# B&R Automation Studio project EFI (part 9)

#### ArcLampGew.var - Local variables
```iecst
VAR CONSTANT
	MAXIMUM_QUANTITY_ALERTS : USINT := 6;
END_VAR
VAR
	data : REFERENCE TO ArcLampGew;
	Client : httpClient := (enable:=FALSE,send:=FALSE,abort:=FALSE,option:=0,pHost:=0,hostPort:=0,method:=httpMETHOD_GET,pUri:=0,pRequestHeader:=0,pRequestData:=0,requestDataLen:=0,pResponseHeader:=0,pResponseData:=0,responseDataSize:=0,pStatistics:=0,pStruct:=0,status:=0,tcpStatus:=0,httpStatus:=0,responseDataLen:=0,phase:=0,_i_state:=0,_i_result:=0,_ident:=0,_oldEnable:=0,_oldAbort:=0,_oldSend:=0,_state:=0,_internal:=0);
	ClientPost : httpClient := (enable:=FALSE,send:=FALSE,abort:=FALSE,option:=0,pHost:=0,hostPort:=0,method:=httpMETHOD_GET,pUri:=0,pRequestHeader:=0,pRequestData:=0,requestDataLen:=0,pResponseHeader:=0,pResponseData:=0,responseDataSize:=0,pStatistics:=0,pStruct:=0,status:=0,tcpStatus:=0,httpStatus:=0,responseDataLen:=0,phase:=0,_i_state:=0,_i_result:=0,_ident:=0,_oldEnable:=0,_oldAbort:=0,_oldSend:=0,_state:=0,_internal:=0);
	Doenable : BOOL := FALSE; (*Enables FUB Instance*)
	Dosend : BOOL := FALSE; (*Sends request on positive edge*)
	Host : STRING[100] := 'localhost';
	Responsedata : STRING[6000] := '';
	Ressource : STRING[80] := '';
	RequestHeader : httpResponseHeader_t;
	RequestHeaderPost : httpResponseHeader_t;
	credentialsFlat : STRING[80];
	CredentialsEncoder : httpEncodeBase64;
	credentialsBase64 : STRING[280];
	authenticationBase : STRING[180];
	strAux : STRING[80];
	JSON_Parse_0 : JSON_Parse;
	dataToParse : STRING[6000] := '';
	sysResp : SystemResp;
	LampsResp : AllLampsResp;
	UvLampsResp : UvStatusResp;
	alertsResp : AlertsLampResp;
	sysRespWrk : SystemResp;
	LampsRespWrk : AllLampsResp;
	UvLampsRespWrk : UvStatusResp;
	alertsRespWrk : AlertsLampResp;
	commsStatus : ArcLampGew_Comms := ARCLG_IDLE;
	commsStatus_copy : ArcLampGew_Comms := ARCLG_IDLE;
	xComsStatusChanged : BOOL;
	commsSubStatus : ArcLampGew_SubComms := ARCLGS_IDLE;
	dataDebug : STRING[1800];
	dataNotFound : STRING[180];
	CurrentState : ArcLampGew_State := ARCLGEW_NOT_INITIALIZED;
	CurrentState_copy : ArcLampGew_State := ARCLGEW_NOT_INITIALIZED;
	xCurrentStateChanged : BOOL;
END_VAR
VAR CONSTANT
	iHistoryLines : USINT := 25;
END_VAR
VAR
	StateHistory : ARRAY[0..iHistoryLines] OF ArcLampGew_State;
	iIndexHistory : USINT;
	iLamp : USINT;
	iAlert : USINT;
	CommsCmdReseted : CommsCommands;
	xAnyLampSelected : BOOL;
	xAnyLampInError : BOOL;
	tonErrorComms : TON;
	tonSendReadSystem : TON;
	tonDelaySendReadSystem : TON;
	resetedAlarms : ArcLampGew_Alarms;
	resetedAlarmsSummary : stEFI_AlarmSummary;
	resetedComsAlarms : ArcLampGew_CommsAlarms;
	xAuxVar : BOOL;
	iLampComs : USINT; (*Variable to define the lamp communicating with. NOT to use in loops*)
	iMaxLampSelected : USINT; (*The maximum selected lamp prepare to workwith*)
	paramURL : httpSetParamUrl;
	RequestDataPost : STRING[180];
	iStatusChanges : UINT;
	iReasonStop : UINT;
	iReasonCritical : UINT;
	iAnyAlarm : UINT;
	iAnyWarning : UINT;
	stEventLog : EventLog_typ;
	reasonSound : UINT;
	arCommsError : AutoResetSound;
	arLampInError1 : AutoResetSound;
	arLampInError2 : AutoResetSound;
	arJam : AutoResetSound;
	iTimesReadLamps : UINT;
	iTimesReadLampsUv : UINT;
	iTimesReadAlerts : UINT;
	iTimesResetAll : UINT;
	iTimesSelectLamp : UINT;
	iTimesDeselectLamp : UINT;
	iTimesStopSelected : UINT;
	iTimesStartSelected : UINT;
	iTimesDeselectAll : UINT;
	iTimesSetPower : UINT;
	iTimesReadSystem : UINT;
	iTimesCommsError : UINT;
	credentialsUser : STRING[80];
	credentialsUserInternal : STRING[80];
	strAuxCredentials : STRING[80];
	iSendClient : UINT;
	iSendPost : UINT;
	lastErrorReseted : ErrorWebServiceData;
	lastCommsError : ErrorWebServiceData;
END_VAR
VAR CONSTANT
	iHistoryCommsLines : USINT := 25;
END_VAR
VAR
	ErrorCommsHistory : ARRAY[0..iHistoryCommsLines] OF ErrorWebServiceData;
	iIndexCommsHistory : USINT;
	UvLampRespAssigWrk : REFERENCE TO UvLampResp;
	tonParsingError : TON;
	tonInputReady : TON;
	tonRetryCommand : TON;
	xResetNeeded : UINT;
	xReadSystemDelay : BOOL;
	iReasonToStop : USINT;
	resetedOuts : ArcLampGew_SignalsOut;
	resetedStatus : ArcLampGew_Status;
END_VAR
```

- Rhino API - Read-Write.postman_collection.json (not shown)

### ArcLampSim.typ
```iecst
TYPE
	ArcLampSimCommands_typ : 	STRUCT
		CreateError : BOOL;
	END_STRUCT;
	ArcLampSim_typ : 	STRUCT
		Commands : ArcLampSimCommands_typ;
	END_STRUCT;
END_TYPE
```

### Program Logical/ExtPack/_Cure/ArcLampGEW/ArcLampSim/ArcLampSim_v1/ArcLampSim (IEC)

#### ArcLampSim.var - Local variables
```iecst
VAR
	SimArcLamp : REFERENCE TO ArcLampSim_typ;
	dataArcLamp : REFERENCE TO ArcLampGew;
	tonTransport : TON;
	tonReady : TON;
	tonDry : TON;
	CommsCmdReseted : CommsCommands;
	tonCommand : TON;
	iIndexLamp : USINT;
	xSimulatingCommand : UINT;
	iSetLampTimes : UINT;
END_VAR
```

### CuringLed.typ
```iecst
TYPE
	CuringLedCheck_enum :
		(
		CHECK_INIT,
		CHECK_READ_CONFIG,
		CHECK_UPDATE_STATUS,
		CHECK_READY,
		CHECK_ERROR
		);
	CuringLedReadingLampUvTime_enum :
		(
		READINGUVTIME_NOT_INIT,
		READINGUVTIME_INIT,
		READINGUVTIME_READING,
		READINGUVTIME_READY,
		READINGUVTIME_ERROR
		);
	CuringLedReadingLampTemp_enum :
		(
		READINGTEMP_NOT_INIT,
		READINGTEMP_INIT,
		READINGTEMP_READING,
		READINGTEMP_READY,
		READINGTEMP_ERROR
		);
	CuringLedDetect_enum :
		(
		DETECTION_NOT_INIT,
		DETECTION_INIT,
		DETECTION_POLLING,
		DETECTION_SAVE_SERIAL_NUMBERS,
		DETECTION_FINISHING_POLLING,
		DETECTION_READ_INTENSITY,
		DETECTION_ASSIGN_POSITION,
		DETECTION_READY,
		DETECTION_ERROR
		);
	CuringLedConfig_enum :
		(
		CONFIGURATION_NOT_INIT,
		CONFIGURATION_INIT,
		CONFIGURATION_PREPARE_LAMP,
		CONFIGURATION_PREPARE_SLM,
		CONFIGURATION_SEND,
		CONFIGURATION_SENDING,
		CONFIGURATION_SENT,
		CONFIGURATION_READ,
		CONFIGURATION_READY
		);
	CuringLedStatus_enum :
		(
		CURINGLED_OFF,
		CURINGLED_INIT,
		CURINGLED_PREPARING,
		CURINGLED_READY,
		CURINGLED_EMITTING,
		CURINGLED_FAULTED
		);
	CuringLed_NitrogenStatus_enum :
		(
		CURINGNITRO_OFF,
		CURINGNITRO_INIT,
		CURINGNITRO_READY,
		CURINGNITRO_FAULT
		);
	CuringLed_ApplicationType_enum :
		( (*Defines application purpose of curing led. May be use to cure ink (white, color) or primer*)
		CURING_APP_UNDEFINED,
		CURING_APP_WHITE, (*White ink*)
		CURING_APP_COLOR, (*Any ink apart from white*)
		CURING_APP_PRIMER (*Varnish*)
		);
	CuringLed_Alarms_typ : 	STRUCT
		xChillerFaulted : BOOL;
		xN2HighFlow : BOOL;
		xN2LowFlow : BOOL;
		xCureSystemFaulted : BOOL; (*gui_q_xAlrOverallCureSystFaulted*)
		xLampsSlmNotConfigured : BOOL;
		xFrontDoorOpened : BOOL; (*Front door is opened. UV light is dangerous*)
		xPowerFailure : BOOL; (*Any power suppliy dc voltage has failed*)
		xSerialNumbersRepeated : BOOL; (*Some lamps has same serial number*)
		xSerialNumbersNotAssigned : BOOL; (*Any lamp has no serial number assigned*)
		xDetectionProcessFailed : BOOL; (*Serial number detection process has failed*)
		Lamps : ARRAY[0..MAX_LAST_CURING_LED_LAMP]OF CuringLed_Lamp_Alarms_typ;
	END_STRUCT;
	CuringLed_Lamp_Alarms_typ : 	STRUCT
		SLMFault : BOOL; (*SLM fault present on LED cure lamp*)
		ThermalFault : BOOL; (*Thermal fault present on LED cure lamp*)
		AnyWarning : BOOL; (*Warning if there is any not needed lamp in error.*)
		StatusFeedbackFault : BOOL; (*Slm status feedback from lamp missing in system status message*)
		xSlmWrongConfiguration : ARRAY[0..20]OF BOOL; (*SLM not configured properly*)
	END_STRUCT;
	CuringLed_Signals_In_typ : 	STRUCT
		xN2HighFlow : BOOL;
		xN2LowFlow : BOOL;
		xPsuDcOk : ARRAY[0..10]OF BOOL;
		xPsuAcOk : ARRAY[0..10]OF BOOL;
		xFrontDoorClosed : BOOL;
		xSafetyEnable : BOOL; (*The Enable signals are active. Do not show alarms related to this if not active*)
	END_STRUCT;
	CuringLed_Signals_Out_typ : 	STRUCT
		xPowerOnLamps : BOOL;
		xRunChiller : BOOL; (*Chiller has just one input named "Run"*)
		xPowerOnNitrogen : BOOL;
	END_STRUCT;
	CuringLed_Signals_typ : 	STRUCT
		Inputs : CuringLed_Signals_In_typ;
		Outputs : CuringLed_Signals_Out_typ;
	END_STRUCT;
	CuringLed_Comms_typ : 	STRUCT
		Ready : BOOL; (*To show the status of the startup process.*)
		ConfigOK : BOOL; (*Lamps SLMs configured*)
		Command : Comms_command_typ;
		Device : DeviceComms_typ;
	END_STRUCT;
	CuringLed_Status_typ : 	STRUCT
		xInstalled : BOOL;
		xEmitting : BOOL;
		DetectionState : CuringLedDetect_enum; (*State of the control*)
		Config : CuringLedConfig_enum; (*State of the control*)
		State : CuringLedStatus_enum; (*Status of the curing led: 0=off, 1=init, 2=ready, 3=emitting, 4=faulted*)
		NitroState : CuringLed_NitrogenStatus_enum;
		ChillerState : ChillerStatus_enum;
		iTotalNumSlms : UINT; (*Total number of slm of the curing bar*)
		xOptimizeCuring : BOOL; (*To cure just the document not the entire board*)
		xCureByStretch : BOOL; (*To configure lamps to cure by stretches*)
		xLampsDetected : BOOL; (*Active when all lamps installed have a serial number associated*)
		xLampsChecked : BOOL; (*Active when check of lamps current configuration match desired configuration*)
		xLampsConfigured : BOOL; (*Active when all lamps have been configured*)
		ManualCommands : CuringLed_ManualCommands_typ;
		iCuringAreaWidth : UINT;
		iCuringAreaOffsetL1 : INT;
		iCuringAreaOffsetL2 : INT;
	END_STRUCT;
	CuringLed_Parameters_typ : 	STRUCT
		xInstalled : BOOL;
		xEnabled : BOOL;
		iLampsQuantity : USINT; (*Total lamps in the CuringLed system. Max 16*)
		Mode : StGeneral_States_Mode;
		AutoMode : stEFI_MachineAutoModes;
		iChillerIndex : INT; (*Index of chiller used by the curing led lamp*)
		iCuringPosition : INT; (*Position of the led lamps bar in cm*)
		iCuringWindow : INT; (*Led lamps width in process direction (in mm). Depends on lamp's model. Alll lamps on same led bar have the same*)
		iDocumentWidth : UINT;
		iDocumentOffsetL1 : INT;
		iDocumentOffsetL2 : INT;
		iMaxCuringAreaWidth : UINT;
		iMaxCuringAreaOffsetL1 : INT;
		iMaxCuringAreaOffsetL2 : INT;
		iMediaWidth : UINT;
		iMediaOffsetL1 : INT;
		iMediaOffsetL2 : INT;
		xDoubleLine : BOOL;
		rBeltCurrentSpeed : REAL;
		rMinCureSpeed : REAL := 1;
		iPowerSuppliesQuantity : USINT; (*Total power supplies used to power all lamps in the curing led bar. Max 10*)
		xWhiteLedBar : BOOL; (*To set this variable to TRUE when curing led bar is used for white color*)
		xCureBySpeed : BOOL; (*Intensity of lamps set depending on machine speed*)
		xSimulationMode : BOOL;
		xOptimizeCuring : BOOL; (*Curing optimitzation required*)
		xCureByStretch : BOOL; (*Curing by stretch mode required*)
		xPhysicalTempFeedback : BOOL; (*When a plc card is installed to read temp from lamp using an AI*)
		iMappingBar : USINT;
		iSlmWidth : USINT := 25;
		CuringApplicationType : CuringLed_ApplicationType_enum;
	END_STRUCT;
	CuringLed_ManualCommands_typ : 	STRUCT
		xNitrogen : BOOL;
		DetectLamps : BOOL;
		ResetPSU : BOOL; (*Reset the PSU to power the Lamps*)
	END_STRUCT;
	CuringLed_Commands_typ : 	STRUCT
		PowerOn : BOOL;
		xDropPower : BOOL; (*Command to set lamps to a lower intensity than defined by curing mode or setpoint written by SW*)
		xRunNitrogenFlow : BOOL; (*Command to active nitrogen flow*)
		xUpdateTempValues : BOOL; (*Update temp values*)
		RunCuring : BOOL; (*When the media to cure is below the lamps*)
		Mute : BOOL; (*command xMute *)
		Reset : BOOL; (*command xReset*)
		Manual : CuringLed_ManualCommands_typ;
	END_STRUCT;
	CuringLed_typ : 	STRUCT
		Signals : CuringLed_Signals_typ;
		Commands : CuringLed_Commands_typ;
		Parameters : CuringLed_Parameters_typ;
		Status : CuringLed_Status_typ;
		Alarms : CuringLed_Alarms_typ;
		AlSummary : stEFI_AlarmSummary; (*Alarms Summary*)
		Comms : CuringLed_Comms_typ;
		Lamp : ARRAY[0..MAX_LAST_CURING_LED_LAMP]OF CuringLed_Lamp_typ;
		parSw : CuringLed_Sw_Parameters_typ;
	END_STRUCT;
	enComms_STEPS :
		(
		FRM_WAIT := 0, (*Defines the wait step*)
		FRM_OPEN := 10, (*Defines Step for FRM_xopen() *)
		FRM_CLEAR_BUFFER := 20, (*Defines Step for FRM_rbuf()*)
		FRM_PREPARE_SENDDATA := 21, (*Defines Step for preparing send data*)
		FRM_WRITE := 22, (*Defines Step for FRM_write()*)
		FRM_RELEASE_SEND_BUFFER := 23, (*Defines Step for FRM_robuf()*)
		FRM_READ := 30, (*Defines Step for FRM_read()*)
		FRM_COPY_RD_DATA := 31, (*Defines Step for storing read data*)
		FRM_RELEASE_READ_BUFFER := 32, (*Defines Step for FRM_rbuf()*)
		FRM_CLOSE := 40, (*Defines Step for FRM_close()*)
		FRM_ERROR := 255 (*Defines Step for Errorhandling*)
		);
	Comms_command_typ : 	STRUCT
		Open : BOOL; (*Open serial port and receive data*)
		Send : BOOL; (*Close serial port*)
		Receive : BOOL; (*Receive data from device*)
		Close : BOOL; (*Close serial port*)
	END_STRUCT;
	DeviceComms_typ : 	STRUCT
		step : enComms_STEPS := (0); (*Step of the Statemachine*)
		receive_data : STRING[800]; (*receive data*)
		send_data : STRING[80]; (*Send data*)
		FRM_xopen_0 : FRM_xopen; (*Functionblock FRM_xopen()*)
		xopenConfig : XOPENCONFIG; (*Configuration Type for FRM_xopen()*)
		FRM_gbuf_0 : FRM_gbuf; (*Functionblock FRM_gbuf()*)
		FRM_robuf_0 : FRM_robuf; (*Functionblock FRM_robuf()*)
		FRM_read_0 : FRM_read; (*Functionblock FRM_read()*)
		FRM_rbuf_0 : FRM_rbuf; (*Functionblock FRM_rbuf()*)
		FRM_write_0 : FRM_write; (*Functionblock FRM_write)*)
		FRM_close_0 : FRM_close; (*Functionblock FRM_close()*)
		DeviceName : STRING[22]; (*Devicename --> serial interface properties*)
	END_STRUCT;
	CuringLed_Lamp_typ : 	STRUCT
		Inputs : CuringLed_Lamp_Inputs_typ;
		Outputs : CuringLed_Lamp_Outputs_typ;
		Parameters : CuringLed_Lamp_Parameters_typ;
		Status : CuringLed_Lamp_Status_typ;
	END_STRUCT;
	CuringLed_Lamp_Status_typ : 	STRUCT
		stUvOnTimeRaw : STRING[10]; (*Total number of minutes that DC power has been applied*)
		rUvOnTime : REAL; (*Total number of minutes that DC power has been applied*)
		rTemp : REAL;
		stSerialNumber : STRING[6];
	END_STRUCT;
	CuringLed_Lamp_Parameters_typ : 	STRUCT
		xInstalled : BOOL := FALSE;
		EnabledByPosition : BOOL := TRUE; (*Enable lamp to be ready for curing depending on its position, board width and offsets*)
		iNumSLM : UINT; (*Number of stretches (slm) in this lamp*)
		iCuringLength : UINT; (*Length of lamp in mm. Per position in lamp's bar (length = cross direction)*)
		xSlmEnable : ARRAY[0..20]OF BOOL; (*SLM to be enabled for each lamp. 1:Must cure, 0: Must not cure*)
		xFullActive : BOOL;
		sSystemStatusFeedback : STRING[300];
		iFirstSlm : INT;
		iLastSlm : INT;
	END_STRUCT;
	CuringLed_Sw_Parameters_typ : 	STRUCT
		IntensitySetPoint : INT; (*Value of the Intensity in percentage. Minimum 10%. gui_i_iUvIntensitySetPointLed1*)
		xEnableDDC : BOOL; (*Enable the DDC functionality*)
		iPreCuringOffset : INT := 0; (*Pre curing offset set by SW in cm*)
		iPostCuringOffset : INT := 0; (*Post curing offset set by SW in cm*)
	END_STRUCT;
	CuringLed_Lamp_Inputs_typ : 	STRUCT
		TemperatureRaw : INT; (*Led temperature value in C.*)
		SLMFault : BOOL; (*SLM fault present on LED cure lamp 1*)
		ThermalFault : BOOL; (*Thermal fault present on LED cure lamp 1*)
	END_STRUCT;
	CuringLed_Lamp_Outputs_typ : 	STRUCT
		IntensityLampApplied : USINT; (*Value of the real intensity setpoint applied to lamp by the PLC*)
		IntensityLampRaw : INT; (*Value of the Intensity in Analog units*)
		EnableLamp : BOOL; (*Enable for each lamp of the curing LED*)
		rTemperature : REAL; (*Lamp  temperature value in C*)
		LampErrorCode : USINT;
		xSlmStatus : ARRAY[0..20]OF BOOL; (*SLM status. Shows SLM is active to cure: 1:On, 0:Off*)
	END_STRUCT;
END_TYPE
```

### CuringLed.var
```iecst
VAR
	iIndexCuringLed : USINT;
END_VAR
```

### Program Logical/ExtPack/_Cure/CuringLedCtrl/CuringLedCtrl_v1/CuringLedCtrl

#### CuringLedCtrlConstants.var
```iecst
VAR CONSTANT
	iSlmWidth : INT := 25;
	StCmdWrite : STRING[2] := 'w ';
	StOff : STRING[2] := 'Of';
	StValueDisableSlm : STRING[2] := ' 0';
	StValueEnableSlm : STRING[2] := ' 1';
	iMaxNumLamps : USINT := 16;
	StCmdEnableSlm : STRING[11] := ' slmenable ';
	StCheckIntensity : STRING[10] := ' intensity';
	StCmdRead : STRING[2] := 'r ';
	StDs : STRING[3] := ' ds';
	StCheckStatus : STRING[4] := ' son'; (*Check if UV is Enabled. [On = UV enabled, Off = UV disabled]*)
	StOn : STRING[2] := 'On';
	StMl : STRING[2] := 'm1';
	BUSY : UINT := 65535; (*Functionblock BUSY status*)
	StCmdDisableAll : STRING[9] := ' slmall 0';
	StCmdEnableAll : STRING[9] := ' slmall 1';
	rCureBySpeedWhiteIntercept : REAL := 14.84;
	rCureBySpeedDefaultIntercept : REAL := 0;
	rCureBySpeedWhiteSlope : REAL := 0.86;
	rCureBySpeedDefaultSlope : REAL := 1.67;
	rLampIntensitySlope : REAL := 327.67;
	StOk : STRING[2] := 'ok';
	StPoll : STRING[4] := 'poll';
	StIntensity : STRING[10] := ' intensity';
	StTemperature : STRING[4] := ' tmp';
	iMaxNumAttempts : INT := 2;
	MaxIntensityCuringBySpeed : USINT := 100;
	MinIntensityCuringBySpeed : USINT := 40;
END_VAR
VAR
	iIntensityAnswerLength : INT := 3;
	iStatusAnswerLength : INT := 2;
END_VAR
```

#### AlarmSound.st
```iecst
ACTION AlarmSound:

	// Alarms reseteable sound management.
	ars_AlrStop.xAlarm:= dataLed.AlSummary.xAlarmStop;
	ars_AlrStop.xSilence:= dataLed.Commands.Mute;
	ars_AlrStop();

	ars_AlrCritical.xAlarm:= dataLed.AlSummary.xAlarmCritical;
	ars_AlrCritical.xSilence:= dataLed.Commands.Mute;
	ars_AlrCritical();

	ars_AlrWarning.xAlarm:= dataLed.AlSummary.xAnyWarning;
	ars_AlrWarning.xSilence:= dataLed.Commands.Mute;
	ars_AlrWarning();

	dataLed.AlSummary.xAlarmSound:= //ars_AlrWarning.xAlarmSound OR
									ars_AlrStop.xAlarmSound OR
									ars_AlrCritical.xAlarmSound;

END_ACTION
```

#### CheckLampsConfig.st
```iecst
ACTION CheckLampsConfig:

	IF (xBoardPositionChanged OR dataLed.Alarms.xPowerFailure OR NOT dataLed.Commands.PowerOn OR EDGEPOS(xConfigurationFailed)) THEN
		CheckStep := CHECK_INIT;
	END_IF

	CASE CheckStep OF

		CHECK_INIT:
			IF dataLed.Status.xLampsConfigured THEN
				iIndexConfigLamps := 1;
				dataLed.Comms.Device.receive_data := '';
				FOR iIndexEraseReceivedData:=1 TO iLampsQuantity DO
					dataLed.Lamp[iIndexConfigLamps].Parameters.sSystemStatusFeedback := '';
				END_FOR
				CheckStep := CHECK_READ_CONFIG;
			END_IF

		CHECK_READ_CONFIG:
			//To set the message string
			ReadLampStatus;

			//To send command to lamp
			dataLed.Comms.Command.Send := TRUE;

			IF (dataLed.Comms.Device.receive_data <> '') THEN
				iSupplySide := 0;
				CheckStep := CHECK_UPDATE_STATUS;
			END_IF

		CHECK_UPDATE_STATUS:
			iNumLampSLM := dataLed.Lamp[iIndexConfigLamps].Parameters.iNumSLM; //Number of lamp's SLMs
			iMinBufferLength := 436 + iNumLampSLM*5; //DELOREAN-1923: Minimum buffer length when lamp gives all slm feedback is: 436+iNumLampSLM*5 (f.e: "1=On ")

			iSupplySide := FIND(dataLed.Comms.Device.receive_data, 'Supply Side');
			xValidStatusReading := iSupplySide>0;
			//IF dataLed.Comms.Device.FRM_read_0.buflng > 500(*iMinBufferLength*) THEN
			IF xValidStatusReading THEN
				iCheckStatusAttempts := 0;
				xSLMStatusRead := TRUE;

				//Saving slms status as lamp parameter
				FindInString := INT_TO_STRING(1);
				strcat(ADR(FindInString),ADR('='));
				iAnswerStringPosition := FIND(dataLed.Comms.Device.receive_data, FindInString);
				dataLed.Lamp[iIndexConfigLamps].Parameters.sSystemStatusFeedback := MID(dataLed.Comms.Device.receive_data, 280, iAnswerStringPosition);

				FOR iIndexConfigSlm:=1 TO iNumLampSLM DO
					CheckSlmStatus;
				END_FOR

				IF xSLMStatusRead THEN
					NextLamp;
				ELSE
					dataLed.Comms.Device.receive_data := '';
					CheckStep := CHECK_READ_CONFIG;
				END_IF

			ELSIF (iCheckStatusAttempts >= iMaxNumAttempts) THEN
				dataLed.Alarms.Lamps[iIndexConfigLamps].StatusFeedbackFault := TRUE;
				NextLamp;

			ELSIF dataLed.Comms.Device.step = FRM_WAIT THEN
				iCheckStatusAttempts := iCheckStatusAttempts + 1;
				dataLed.Comms.Device.receive_data := '';
				CheckStep := CHECK_READ_CONFIG;
			END_IF

		CHECK_READY:

	END_CASE

	dataLed.Comms.Device.send_data := StMessage; //To assign Message to dataled comms struct
	dataLed.Status.xLampsChecked := CheckStep = CHECK_READY;

END_ACTION

//Telegrams to be sent to curing led devices//
//To enable all slm in the lamp
ACTION ReadLampStatus:
	//To define the string to be sent to the lamp
	StMessage := StCmdRead;
	//strcat: Used to link (concat) several strings
	strcat(ADR(StMessage), ADR(dataLed.Lamp[iIndexConfigLamps].Status.stSerialNumber));
	strcat(ADR(StMessage), ADR(StMl));
	strcat(ADR(StMessage), ADR(StDs));
	//dataLed.Comms.Device.send_data := StMessage; //To assign Message to dataled comms struct

	iAnswerStringLength := 2;

	//This is the data received when reading status of a led. SLM status shown for a lamp with all SLM disabled:
	(*
	Product..........: Fire_Line_400_300, s/n 414086m1
	Firmware Ver.....: 01.02
	Log Entries......: 1020
	SLM Enables......:
	Supply Side 1=Off 2=Off 3=Off 4=Off 5=Off 6=Off 7=Off 8=Off 9=Off 10=Off 11=Off 12=Off Return Side
	SW-Disable Low.....: High
	SW-Enable High...: Low
	Global Control...: DB15
	Intensity........: 100
	Temperature......: 36.4
	Inputvolt........: 49.8
	Thermal Switch...: Enabled
	*)
END_ACTION

ACTION NextLamp:

	//Erasing buffer and going to next lamp
	iIndexConfigLamps := iIndexConfigLamps + 1;
	IF iIndexConfigLamps <= iLampsQuantity THEN
		dataLed.Comms.Device.receive_data := '';
		CheckStep := CHECK_READ_CONFIG;
	ELSE
		CheckStep := CHECK_READY;
	END_IF
END_ACTION

ACTION CheckSlmStatus:
	FindInString := INT_TO_STRING(iIndexConfigSlm);
	strcat(ADR(FindInString),ADR('='));
	iAnswerStringPosition := FIND(dataLed.Comms.Device.receive_data, FindInString);
	IF iIndexConfigSlm<10 THEN iAnswerStringPosition := iAnswerStringPosition+2; ELSE iAnswerStringPosition := iAnswerStringPosition+3; END_IF //X=On/Off
	StAnswer := MID(dataLed.Comms.Device.receive_data, iAnswerStringLength, iAnswerStringPosition);

	IF (StAnswer = StOn) THEN
		dataLed.Lamp[iIndexConfigLamps].Outputs.xSlmStatus[iIndexConfigSlm]:=TRUE;
	ELSIF (StAnswer = StOff) THEN
		dataLed.Lamp[iIndexConfigLamps].Outputs.xSlmStatus[iIndexConfigSlm]:=FALSE;
	ELSE
		xSLMStatusRead := FALSE;
	END_IF
END_ACTION
```

#### CheckParameters.st
```iecst
ACTION CheckParameters:

	iLampsQuantity := LIMIT(1,dataLed.Parameters.iLampsQuantity,iMaxNumLamps);
	iPowerSuppliesQuantity := LIMIT(1,dataLed.Parameters.iPowerSuppliesQuantity,6);

	FOR iIndexCuring:=1 TO iLampsQuantity DO
		dataLed.parSw.IntensitySetPoint:=LIMIT(10, dataLed.parSw.IntensitySetPoint, 100);
		dataLed.Lamp[iIndexCuring].Parameters.xInstalled := TRUE;
	END_FOR

	//Assigning parameters of curing area
	IF NOT dataLed.Status.xOptimizeCuring THEN
		dataLed.Status.iCuringAreaWidth := dataLed.Parameters.iMediaWidth;
		dataLed.Status.iCuringAreaOffsetL1 := dataLed.Parameters.iMediaOffsetL1;
		dataLed.Status.iCuringAreaOffsetL2 := dataLed.Parameters.iMediaOffsetL2;
	ELSE
		//Optimize curing will be active when EHD is enabled so plc does not have to consider metal bands overlap with to not burn it.
		//Document width has to be smaller than (MediaWidth- 2*Overlap). Document width is managed by SW
		dataLed.Status.iCuringAreaWidth := dataLed.Parameters.iDocumentWidth;
		dataLed.Status.iCuringAreaOffsetL1 := dataLed.Parameters.iDocumentOffsetL1;
		dataLed.Status.iCuringAreaOffsetL2 := dataLed.Parameters.iDocumentOffsetL2;
	END_IF

	dataLed.Status.iCuringAreaWidth := MIN(dataLed.Status.iCuringAreaWidth, dataLed.Parameters.iMaxCuringAreaWidth);
	dataLed.Status.iCuringAreaOffsetL1 := MAX(dataLed.Status.iCuringAreaOffsetL1, dataLed.Parameters.iMaxCuringAreaOffsetL1);
	dataLed.Status.iCuringAreaOffsetL2 := MIN(dataLed.Status.iCuringAreaOffsetL2, dataLed.Parameters.iMaxCuringAreaOffsetL2);

	//This action must be executed just once.
	IF iTotalNumSlms<=0 THEN
		//To sum all slm in the curing led bar. Depends on number of lamps and their width
		FOR iIndexEnableLamps:=1 TO iLampsQuantity DO
			dataLed.Lamp[iIndexEnableLamps].Parameters.iNumSLM := (dataLed.Lamp[iIndexEnableLamps].Parameters.iCuringLength/iSlmWidth);
			iTotalNumSlms :=  iTotalNumSlms + dataLed.Lamp[iIndexEnableLamps].Parameters.iNumSLM;
		END_FOR

		iTotalNumSlms :=  MIN(iTotalNumSlms, 100);
		dataLed.Status.iTotalNumSlms := iTotalNumSlms;
	END_IF

END_ACTION
```

#### CommsManager.st
```iecst
ACTION CommsManager:

	//To disable functions and open again when a READ command seems to be on hold to much time
	tonOpenPort.IN:= (dataLed.Comms.Device.step = FRM_READ);
	tonOpenPort.PT := T#10s;
	tonOpenPort();

	dataLed.Comms.Command.Open := tonOpenPort.Q;

	IF dataLed.Comms.Command.Open THEN																(*command for sender activation*)
		DisableFunctions;
		dataLed.Comms.Device.step := FRM_OPEN;

	ELSIF dataLed.Comms.Command.Close THEN															(*command for sender activation*)
		DisableFunctions;
		dataLed.Comms.Device.step := FRM_CLOSE;
	END_IF

	CASE dataLed.Comms.Device.step OF

		FRM_WAIT:
			IF dataLed.Comms.Command.Send THEN													(*command for sender activation*)
				dataLed.Comms.Device.step := FRM_OPEN;
			ELSIF dataLed.Comms.Command.Receive THEN											(*command for sender activation*)
				dataLed.Comms.Device.step := FRM_READ;
			END_IF

		FRM_OPEN:
			DisableFunctions;

			(*Parameters for FRM_xopen()*)
			dataLed.Comms.Device.FRM_xopen_0.enable := TRUE;

			dataLed.Comms.Device.FRM_xopen_0.device := ADR(dataLed.Comms.Device.DeviceName);
			dataLed.Comms.Device.FRM_xopen_0.mode := ADR('/PHY=RS485 /BD=57600 /DB=8 /PA=N /SB=1'); (*Modestring --> specifies the seria operation mode*)
			dataLed.Comms.Device.FRM_xopen_0.config := ADR(dataLed.Comms.Device.xopenConfig);		(*Additional Parameters, optional*)

			(*Additional Parameters for FRM_xopen()*)
			dataLed.Comms.Device.xopenConfig.idle := 10;											//Idle time between two characters
			dataLed.Comms.Device.xopenConfig.delimc := 0;											//activate two delimeters
			dataLed.Comms.Device.xopenConfig.delim[0] := 0; 										//CR - carridge return -> dec 13
			dataLed.Comms.Device.xopenConfig.delim[1] := 0; 										//LF - line feed -> dec 10
			dataLed.Comms.Device.xopenConfig.tx_cnt := 1;											//number of transmit buffers
			dataLed.Comms.Device.xopenConfig.rx_cnt := 1; 											//number of receive buffers
			dataLed.Comms.Device.xopenConfig.tx_len := 80; 											//length of transmit buffers
			dataLed.Comms.Device.xopenConfig.rx_len := 800; 										//lenght of receive buffers
			dataLed.Comms.Device.xopenConfig.argc := 0;												//activate additional options
			dataLed.Comms.Device.xopenConfig.argv := 0;												//parameters for additional options (check help)
			dataLed.Comms.Device.FRM_xopen_0();														//call the FRM_xopen() function

			xCommsOpened := dataLed.Comms.Device.FRM_xopen_0.status = 0;
			xOpeningComms := dataLed.Comms.Device.FRM_xopen_0.status = BUSY;

			IF dataLed.Comms.Device.FRM_xopen_0.status <> ERR_FUB_BUSY AND dataLed.Comms.Device.FRM_xopen_0.status <> ERR_FUB_ENABLE_FALSE THEN
				IF dataLed.Comms.Device.FRM_xopen_0.status = ERR_OK THEN
					dataLed.Comms.Device.step := FRM_CLEAR_BUFFER;
				ELSE
					dataLed.Comms.Device.step := FRM_ERROR;
				END_IF
			END_IF

		(*aquire sendbuffer for FRM_WRITE*)
		FRM_CLEAR_BUFFER:
			dataLed.Comms.Device.FRM_gbuf_0.enable := TRUE;
			dataLed.Comms.Device.FRM_gbuf_0.ident := dataLed.Comms.Device.FRM_xopen_0.ident;
			dataLed.Comms.Device.FRM_gbuf_0();																	(*call the FRM_gbuf() function*)

			xBufferCleared := dataLed.Comms.Device.FRM_gbuf_0.status = 0;
			xClearingBuffer := dataLed.Comms.Device.FRM_gbuf_0.status = BUSY;

			IF dataLed.Comms.Device.FRM_gbuf_0.status <> ERR_FUB_BUSY AND dataLed.Comms.Device.FRM_gbuf_0.status <> ERR_FUB_ENABLE_FALSE THEN
				IF dataLed.Comms.Device.FRM_gbuf_0.status = ERR_OK THEN
					memset(dataLed.Comms.Device.FRM_gbuf_0.buffer,0,dataLed.Comms.Device.FRM_gbuf_0.buflng);		//clear sendbuffer
					dataLed.Comms.Device.step := FRM_PREPARE_SENDDATA;
				ELSE
					dataLed.Comms.Device.step := FRM_ERROR;
				END_IF
			END_IF

		(*prepare senddata, copy data to sendbuffer*)
		FRM_PREPARE_SENDDATA:
			send_data := dataLed.Comms.Device.send_data;
			strcat(ADR(send_data),ADR('$R$L'));
			strcpy(dataLed.Comms.Device.FRM_gbuf_0.buffer,ADR(send_data));					(*copy senddata to sendbuffer*)

			dataLed.Comms.Device.step := FRM_WRITE;																(*--> next step*)

		(*write data to interface*)
		FRM_WRITE:
			(*Parameters for FRM_write()*)
			dataLed.Comms.Device.FRM_write_0.enable := TRUE;
			dataLed.Comms.Device.FRM_write_0.ident := dataLed.Comms.Device.FRM_xopen_0.ident;					(*ident from FRM_xopen()*)
			dataLed.Comms.Device.FRM_write_0.buffer := dataLed.Comms.Device.FRM_gbuf_0.buffer;					(*sendbuffer*)
			dataLed.Comms.Device.FRM_write_0.buflng := strlen(ADR(send_data));								(*net length of senddata*)

			dataLed.Comms.Device.FRM_write_0();																	(*call the FRM_write() function*)

			xBufferSent := dataLed.Comms.Device.FRM_write_0.status = 0;
			xSendingBuffer := dataLed.Comms.Device.FRM_write_0.status = BUSY;

			IF dataLed.Comms.Device.FRM_write_0.status <> ERR_FUB_BUSY AND dataLed.Comms.Device.FRM_write_0.status <> ERR_FUB_ENABLE_FALSE THEN
				IF dataLed.Comms.Device.FRM_write_0.status = ERR_OK THEN
					dataLed.Comms.Device.step := FRM_RELEASE_SEND_BUFFER;
				ELSE
					dataLed.Comms.Device.step := FRM_ERROR;
				END_IF
			END_IF

		(*release sendbuffer in case of no successful write operation*)
		FRM_RELEASE_SEND_BUFFER:
			dataLed.Comms.Device.FRM_robuf_0.enable := TRUE;
			dataLed.Comms.Device.FRM_robuf_0.buffer := dataLed.Comms.Device.FRM_gbuf_0.buffer;					(*sendbuffer*)
			dataLed.Comms.Device.FRM_robuf_0.buflng := dataLed.Comms.Device.FRM_gbuf_0.buflng;					(*buffer length*)
			dataLed.Comms.Device.FRM_robuf_0.ident := dataLed.Comms.Device.FRM_xopen_0.ident;					(*ident open*)
			dataLed.Comms.Device.FRM_robuf_0();																	(*call the FRM_robuf() function*)

			xBufferSendReleased := dataLed.Comms.Device.FRM_robuf_0.status = 0;
			xReleasingSendBuffer := dataLed.Comms.Device.FRM_robuf_0.status = BUSY;

			IF dataLed.Comms.Device.FRM_robuf_0.status <> ERR_FUB_BUSY AND dataLed.Comms.Device.FRM_robuf_0.status <> ERR_FUB_ENABLE_FALSE THEN
				IF dataLed.Comms.Device.FRM_robuf_0.status = ERR_OK THEN
					dataLed.Comms.Device.step := FRM_READ;
				ELSE
					dataLed.Comms.Device.step := FRM_ERROR;
				END_IF
			END_IF

		(*read data from serial interface*)
		FRM_READ:
			dataLed.Comms.Device.FRM_read_0.enable := TRUE;
			dataLed.Comms.Device.FRM_read_0.ident := dataLed.Comms.Device.FRM_xopen_0.ident;
			dataLed.Comms.Device.FRM_read_0();																	(*call the FRM_read() function*)

			xBufferRead := dataLed.Comms.Device.FRM_read_0.status = 0;
			xReadBufferNoInput := dataLed.Comms.Device.FRM_read_0.status = frmERR_NOINPUT;
			xReadBufferInputError := dataLed.Comms.Device.FRM_read_0.status = frmERR_INPUTERROR;

			IF dataLed.Comms.Device.FRM_read_0.status <> ERR_FUB_BUSY AND dataLed.Comms.Device.FRM_read_0.status <> ERR_FUB_ENABLE_FALSE THEN
				IF dataLed.Comms.Device.FRM_read_0.status = ERR_OK THEN
					dataLed.Comms.Device.step := FRM_COPY_RD_DATA;
				ELSIF  dataLed.Comms.Device.FRM_read_0.status = frmERR_NOINPUT THEN
					dataLed.Comms.Device.step := FRM_READ;
				ELSIF dataLed.Comms.Device.FRM_read_0.status = frmERR_INPUTERROR THEN
					dataLed.Comms.Device.step := FRM_RELEASE_READ_BUFFER;
				ELSE
					dataLed.Comms.Device.step := FRM_ERROR;
				END_IF
			END_IF

		(*copy data out of the receive buffer*)
		FRM_COPY_RD_DATA:
			memset(ADR(dataLed.Comms.Device.receive_data),0,SIZEOF(dataLed.Comms.Device.receive_data));										(*clear read_data buffer*)
			memcpy(ADR(dataLed.Comms.Device.receive_data),dataLed.Comms.Device.FRM_read_0.buffer,dataLed.Comms.Device.FRM_read_0.buflng);   (*copy and evaluate read data*)
			dataLed.Comms.Device.step := FRM_RELEASE_READ_BUFFER;																			(*release read buffer*)

		(*release readbuffer*)
		FRM_RELEASE_READ_BUFFER:
			(*Parameters for FRM_rbuf()*)
			dataLed.Comms.Device.FRM_rbuf_0.enable := TRUE;
			dataLed.Comms.Device.FRM_rbuf_0.ident := dataLed.Comms.Device.FRM_xopen_0.ident;					(*ident from FRM_xopen()*)
			dataLed.Comms.Device.FRM_rbuf_0.buffer := dataLed.Comms.Device.FRM_read_0.buffer;					(*read buffer*)
			dataLed.Comms.Device.FRM_rbuf_0.buflng := dataLed.Comms.Device.FRM_read_0.buflng;					(*length of sendbuffer*)
			dataLed.Comms.Device.FRM_rbuf_0();																	(*call the FRM_rbuf() function*)

			xBufferReadReleased := dataLed.Comms.Device.FRM_rbuf_0.status = 0;
			xReleasingReadBuffer := dataLed.Comms.Device.FRM_rbuf_0.status = BUSY;
			xBufferReadInvalid := dataLed.Comms.Device.FRM_rbuf_0.status = frmERR_INVALIDBUFFER;

			IF dataLed.Comms.Device.FRM_rbuf_0.status <> ERR_FUB_BUSY AND dataLed.Comms.Device.FRM_rbuf_0.status <> ERR_FUB_ENABLE_FALSE THEN
				IF dataLed.Comms.Device.FRM_rbuf_0.status = ERR_OK THEN
					dataLed.Comms.Device.step := FRM_CLOSE;
				ELSIF dataLed.Comms.Device.FRM_rbuf_0.status = frmERR_INVALIDBUFFER THEN
					dataLed.Comms.Device.step := FRM_READ;
				ELSE
					dataLed.Comms.Device.step := FRM_ERROR;
				END_IF
			END_IF

		(*close the interface*)
		FRM_CLOSE:
			DisableFunctions;

			dataLed.Comms.Device.FRM_close_0.enable := TRUE;
			dataLed.Comms.Device.FRM_close_0.ident := dataLed.Comms.Device.FRM_xopen_0.ident;	(*ident from FRM_xopen()*)
			dataLed.Comms.Device.FRM_close_0();													(*call the FRM_close() function*)

			xCommsClosed := dataLed.Comms.Device.FRM_close_0.status = 0;
			xClosingComms := dataLed.Comms.Device.FRM_close_0.status = BUSY;

			IF dataLed.Comms.Device.FRM_close_0.status <> ERR_FUB_BUSY AND dataLed.Comms.Device.FRM_close_0.status <> ERR_FUB_ENABLE_FALSE THEN
				IF dataLed.Comms.Device.FRM_close_0.status = ERR_OK THEN
					dataLed.Comms.Device.step := FRM_WAIT;
				ELSE
					dataLed.Comms.Device.step := FRM_ERROR;
				END_IF
			END_IF

		(*error handling*)
		FRM_ERROR:
			DisableFunctions;
			dataLed.Comms.Device.step := FRM_WAIT;  (*not implementet yet, check help for error codes*)

	END_CASE

	//Store the history OF the error code TO easy the debug
	IF dataLed.Comms.Device.step<>StateHistory[0] THEN
		FOR iIndexHistory:=iHistoryLines TO 1 BY -1 DO
			StateHistory[iIndexHistory]:=StateHistory[iIndexHistory-1];
		END_FOR
		StateHistory[0]:=dataLed.Comms.Device.step;
	END_IF

	//Comms commands
	dataLed.Comms.Command := CommsCommandsReset;

END_ACTION

ACTION DisableFunctions:
	dataLed.Comms.Device.FRM_close_0.enable := FALSE;
	dataLed.Comms.Device.FRM_gbuf_0.enable := FALSE;
	dataLed.Comms.Device.FRM_rbuf_0.enable := FALSE;
	dataLed.Comms.Device.FRM_read_0.enable := FALSE;
	dataLed.Comms.Device.FRM_robuf_0.enable := FALSE;
	dataLed.Comms.Device.FRM_write_0.enable := FALSE;
	dataLed.Comms.Device.FRM_xopen_0.enable := FALSE;
END_ACTION
```

#### ConfigureLamps.st
```iecst
ACTION ConfigureLamps:

	IF dataLed.Alarms.xPowerFailure OR NOT dataLed.Commands.PowerOn THEN ConfigCtrl := CONFIGURATION_NOT_INIT; END_IF
	IF xBoardPositionChanged OR EDGEPOS(xConfigurationFailed) THEN ConfigCtrl := CONFIGURATION_INIT; END_IF

	CASE ConfigCtrl OF

		CONFIGURATION_NOT_INIT:

		CONFIGURATION_INIT:
			iIndexConfigLamps := 1;
			iIndexConfigSlm := 0;
			ConfigCtrl := CONFIGURATION_PREPARE_LAMP;

		CONFIGURATION_PREPARE_LAMP:
			//To evaluate only lamps that are going to be active (EnabledByPosition)
			IF NOT dataLed.Lamp[iIndexConfigLamps].Parameters.EnabledByPosition THEN
				DisableAllSlm;
			ELSE
				//To enable all SLM by default
				EnableAllSlm;
			END_IF
			ConfigCtrl := CONFIGURATION_SEND;

		CONFIGURATION_PREPARE_SLM:
			iNumLampSLM := dataLed.Lamp[iIndexConfigLamps].Parameters.iNumSLM; //Number of lamp's SLMs
			IF iIndexConfigSlm<=iNumLampSLM THEN
				//An active lamp might be full used or just use some SLMs
				IF (NOT dataLed.Lamp[iIndexConfigLamps].Parameters.xSlmEnable[iIndexConfigSlm]) THEN
					StIndex := INT_TO_STRING(iIndexConfigSlm);
					DisableSlm;
				END_IF
				ConfigCtrl := CONFIGURATION_SEND;
			ELSE
				iIndexConfigSlm := 0; //1;
				ConfigCtrl := CONFIGURATION_SENT;
			END_IF

		CONFIGURATION_SEND:
			dataLed.Comms.Command.Send := TRUE;
			ConfigCtrl := CONFIGURATION_SENDING;

		CONFIGURATION_SENDING:
			IF (StAnswer = StGoodAnswer) THEN
				IF (dataLed.Lamp[iIndexConfigLamps].Parameters.xFullActive OR NOT dataLed.Lamp[iIndexConfigLamps].Parameters.EnabledByPosition) THEN
					ConfigCtrl := CONFIGURATION_SENT;
				ELSE
					ConfigCtrl := CONFIGURATION_PREPARE_SLM;
					iIndexConfigSlm := iIndexConfigSlm + 1;
				END_IF
				dataLed.Comms.Device.receive_data := '';
			ELSIF dataLed.Comms.Device.step = FRM_WAIT THEN
				ConfigCtrl := CONFIGURATION_SEND;
			END_IF

		CONFIGURATION_SENT:
			iIndexConfigLamps := iIndexConfigLamps + 1;
			IF iIndexConfigLamps > iLampsQuantity THEN
				ConfigCtrl := CONFIGURATION_READY;
			ELSE
				ConfigCtrl := CONFIGURATION_PREPARE_LAMP;
			END_IF

		CONFIGURATION_READY:

	END_CASE

	dataLed.Comms.Device.send_data := StMessage; //To assign Message to dataled comms struct
	StAnswer := MID(dataLed.Comms.Device.receive_data, iAnswerStringLength, iAnswerStringPosition);
	dataLed.Status.xLampsConfigured := ConfigCtrl = CONFIGURATION_READY;
	dataLed.Status.Config := ConfigCtrl;

END_ACTION

//Telegrams to be sent to curing led devices//
//To enable all slm in the lamp
ACTION EnableAllSlm:
	//To define the string to be sent to the lamp
	StMessage := StCmdWrite;
	//strcat: Used to link (concat) several strings
	strcat(ADR(StMessage), ADR(dataLed.Lamp[iIndexConfigLamps].Status.stSerialNumber));
	strcat(ADR(StMessage), ADR(StMl));
	strcat(ADR(StMessage), ADR(StCmdEnableAll));

	//Devices answers "ok"
	StGoodAnswer := StOk;
	iAnswerStringPosition := 1;
	iAnswerStringLength := 2;
END_ACTION

//To disable all slm in the lamp
ACTION DisableAllSlm:
	//To define the string to be sent to the lamp
	StMessage := StCmdWrite;
	//strcat: Used to link (concat) several strings
	strcat(ADR(StMessage), ADR(dataLed.Lamp[iIndexConfigLamps].Status.stSerialNumber));
	strcat(ADR(StMessage), ADR(StMl));
	strcat(ADR(StMessage), ADR(StCmdDisableAll));

	//Devices answers "ok"
	StGoodAnswer := StOk;
	iAnswerStringPosition := 1;
	iAnswerStringLength := 2;
END_ACTION

//To enable an specific slm in the lamp
ACTION EnableSlm:
	//To define the string to be sent to the lamp
	StMessage := StCmdWrite;
	//strcat: Used to link (concat) several strings
	strcat(ADR(StMessage), ADR(dataLed.Lamp[iIndexConfigLamps].Status.stSerialNumber));
	strcat(ADR(StMessage), ADR(StMl));
	strcat(ADR(StMessage), ADR(StCmdEnableSlm));
	strcat(ADR(StMessage), ADR(StIndex));
	strcat(ADR(StMessage), ADR(StValueEnableSlm));

	//Device answers "SLMxx=On" when DisableSlm command is sent, where xx is SLM Index, so:
	StGoodAnswer := StOn;
	IF iIndexConfigSlm<10 THEN iAnswerStringPosition := 6; ELSE iAnswerStringPosition := 7; END_IF
	iAnswerStringLength := 2;
END_ACTION

//To disable an specific slm in the lamp
ACTION DisableSlm:
	//To define the string to be sent to the lamp
	StMessage := StCmdWrite;
	//strcat: Used to link (concat) several strings
	strcat(ADR(StMessage), ADR(dataLed.Lamp[iIndexConfigLamps].Status.stSerialNumber));
	strcat(ADR(StMessage), ADR(StMl));
	strcat(ADR(StMessage), ADR(StCmdEnableSlm));
	strcat(ADR(StMessage), ADR(StIndex));
	strcat(ADR(StMessage), ADR(StValueDisableSlm));

	//Device answers "SLMxx=Off" when DisableSlm command is sent, where xx is SLM Index, so:
	StGoodAnswer := StOff;
	IF iIndexConfigSlm<10 THEN iAnswerStringPosition := 6; ELSE iAnswerStringPosition := 7; END_IF
	iAnswerStringLength := 2;
END_ACTION
```

#### EnableLamps.st
```iecst
ACTION EnableLamps:
	//Enabling lamps to be activated depending on media width, offset register and line mode (single or 2up)
	iLampPosition := 0;

		IF NOT dataLed.Parameters.xDoubleLine THEN

			//							FEEDER/PRIMER						//
			//																//
			//////////////////////////////////////////////////////////////////
			//User side											//Back side //
			//					  											//
			//								"N" iLampPosition				//
			//----------------------------------------------->|				//
			//[[	1 	  ]][[	...	 ]][[	...	 ]][[	...	 ]][[	 N 	 ]]	//
			//			   ||		  ||	 0	  ||		  ||			//
			//					  			 |								//
			//					  			 |								//
			//			OffsetL1(-)<---------|--------->(+)					//
			//			////////////////////////////////////////////		//
			//			////////////////////////////////////////////		//
			//			////////////////////////////////////////////		//
			//			////////////////////////////////////////////		//
			//			////////////////////////////////////////////		//
			//			////////////////////////////////////////////		//
			//			////////////////////////////////////////////		//
			//			////////////////////////////////////////////		//
			//			|<-------		MediaWidth			------>|		//
			//								 								//
			//iBoardInitPos													//
			//--------->|													//
			//									iBoardFinalPosition			//
			//---------------------------------------------------->|		//
			//////////////////////////////////////////////////////////////////
			//																//
			//							DRYER/STACKER						//

			iBoardInitPosition := MAX(0, iCenterPosition + dataLed.Status.iCuringAreaOffsetL1);
			iBoardFinalPosition := MIN(iTotalWidth, iBoardInitPosition + dataLed.Status.iCuringAreaWidth);
			FOR iIndexEnableLamps:=1 TO iLampsQuantity DO
				iLampPosition := iLampPosition + dataLed.Lamp[iIndexEnableLamps-1].Parameters.iCuringLength;
				dataLed.Lamp[iIndexEnableLamps].Parameters.EnabledByPosition := (iBoardInitPosition < (iLampPosition + dataLed.Lamp[iIndexEnableLamps].Parameters.iCuringLength)) AND
																				(iLampPosition < iBoardFinalPosition);
			END_FOR

		ELSE
			//							FEEDER/PRIMER						//
			//																//
			//////////////////////////////////////////////////////////////////
			//User side											//Back side //
			//					  											//
			//								"N" iLampPosition				//
			//----------------------------------------------->|				//
			//[[	1 	  ]][[	...	 ]][[	...	 ]][[	...	 ]][[	 N 	 ]]	//
			//			   ||		  ||	0	  ||		  ||			//
			//		/////////////////		|	/////////////////			//
			//		/////////////////		|	/////////////////			//
			//		/////////////////		|	/////////////////			//
			//		/////////////////		|	/////////////////			//
			//		/////////////////		|	/////////////////			//
			//		/////////////////		|	/////////////////			//
			//		/////////////////		|	/////////////////			//
			//		/////////////////		|	/////////////////			//
			//		|<- MediaWidth->|		|	|<- MediaWidth->|			//
			//								|								//
			//	iRegisterOffsetL1(-)|<------|-->|iRegisterOffsetL2(+)		//
			//								|								//
			//																//
			//iBoardInitPos													//
			//----->|														//
			//								iBoardFinalPosition				//
			//-------------------------------------------------->|			//
			//								 								//
			//////////////////////////////////////////////////////////////////
			//																//
			//							DRYER/STACKER						//

			iBoardInitPosition := MAX(0,iCenterPosition + dataLed.Status.iCuringAreaOffsetL1);
			iBoardFinalPosition := MIN(iTotalWidth, iCenterPosition + dataLed.Status.iCuringAreaOffsetL2 + dataLed.Status.iCuringAreaWidth);
			FOR iIndexEnableLamps:=1 TO iLampsQuantity DO
				iLampPosition := iLampPosition + dataLed.Lamp[iIndexEnableLamps-1].Parameters.iCuringLength;
				dataLed.Lamp[iIndexEnableLamps].Parameters.EnabledByPosition := (iBoardInitPosition < (iLampPosition + dataLed.Lamp[iIndexEnableLamps].Parameters.iCuringLength)) AND
																				(iLampPosition<iBoardFinalPosition);
			END_FOR

		END_IF

END_ACTION

ACTION MemoBoardParameters:
	iPreviousWidth := dataLed.Status.iCuringAreaWidth;
	iPreviousOffsetRegisterL1 := dataLed.Status.iCuringAreaOffsetL1;
	iPreviousOffsetRegisterL2 := dataLed.Status.iCuringAreaOffsetL2;
END_ACTION
```

#### LedsCuringWidthCalculation.st
```iecst
ACTION StretchesCalculation:

	//Disabling all curing led bar's SLMs
	FOR iIndexEnableSlm:=0 TO iTotalNumSlms DO
		xCuringLedSlms[iIndexEnableSlm] := FALSE;
	END_FOR

	//DELOREAN-1778: To set printer's center
	iTotalWidth := iTotalNumSlms*iSlmWidth;
	iCenterPosition := REAL_TO_INT(iTotalWidth/2);

END_ACTION

ACTION SingleLineCalculation:
	//To caculate first SLM of the total curing led bar SLMs
	rFirstCuringBarSlmL1 := INT_TO_REAL(iCenterPosition + dataLed.Status.iCuringAreaOffsetL1)/iSlmWidth;
	pInteger := ADR(rInteger);
	rMantissa := modf(rFirstCuringBarSlmL1, pInteger);

	iFirstCuringBarSlmL1 := REAL_TO_UINT(rFirstCuringBarSlmL1);
	IF rMantissa = 0.0 THEN iFirstCuringBarSlmL1 := iFirstCuringBarSlmL1 + 1; END_IF

	//To caculate last SLM of the total curing led bar SLMs
	rLastCuringBarSlmL1 := (UINT_TO_REAL(iCenterPosition + dataLed.Status.iCuringAreaOffsetL1 + dataLed.Status.iCuringAreaWidth)/INT_TO_REAL(iSlmWidth));
	pInteger := ADR(rInteger);
	rMantissa := modf(rLastCuringBarSlmL1, pInteger);

	iLastCuringBarSlmL1 := REAL_TO_UINT(rInteger);
	IF rMantissa > 0.0 THEN iLastCuringBarSlmL1 := iLastCuringBarSlmL1 + 1; END_IF
	iLastCuringBarSlmL1 := LIMIT(iFirstCuringBarSlmL1, iLastCuringBarSlmL1, iTotalNumSlms);

	//Activating curing led bar's SLMs
	FOR iIndexEnableSlm:=iFirstCuringBarSlmL1 TO iLastCuringBarSlmL1 DO
		xCuringLedSlms[iIndexEnableSlm] := TRUE;
	END_FOR

	//To enable lamps stretches
	iLastLampSLM := 0;
	FOR iIndexEnableLamps:=1 TO iLampsQuantity DO
		iNumLampSLM := dataLed.Lamp[iIndexEnableLamps].Parameters.iNumSLM; //Number of lamp's SLMs

		//Lamp's first SLM of array "xCuringLedSlms" which considers all SLM in the curing led bar
		iFirstLampSLM := iLastLampSLM + 1;
		iLastLampSLM := iLastLampSLM + dataLed.Lamp[iIndexEnableLamps].Parameters.iNumSLM;

		dataLed.Lamp[iIndexEnableLamps].Parameters.iFirstSlm := iFirstLampSLM;
		dataLed.Lamp[iIndexEnableLamps].Parameters.iLastSlm := iLastLampSLM;

		dataLed.Lamp[iIndexEnableLamps].Parameters.xFullActive := TRUE;

		//Calculating slm mirrored to indexSlm. So xCuringLedSlms starts counting from user side to drive side. But lamps are mechanically assemblied in a reverse way, here an image to understand:

		//xCuringLedSlms[x]	  1						  14  15					  28  29					  42  43					  56
		//Lamp's slm index	  14					   1  14					   1  14					   1  14					   1
							//							//							//							//							//
		//FRONT/USER SIDE//	//			1				//			2				//			3				//			4				//		//REAR/WALKWAY SIDE//
							//							//							//							//							//
							//////////////////////////////////////////////////////////////////////////////////////////////////////////////////

		FOR iIndexEnableSlm:=1 TO iNumLampSLM DO
			iMirrorSlm := iLastLampSLM - iIndexEnableSlm + 1;
			dataLed.Lamp[iIndexEnableLamps].Parameters.xSlmEnable[iIndexEnableSlm] := xCuringLedSlms[iMirrorSlm];

			IF (NOT dataLed.Lamp[iIndexEnableLamps].Parameters.xSlmEnable[iIndexEnableSlm]) THEN
				dataLed.Lamp[iIndexEnableLamps].Parameters.xFullActive := FALSE;
			END_IF
		END_FOR
	END_FOR

END_ACTION

ACTION DoubleLineCalculation:

	///////////		L1		///////////
	rFirstCuringBarSlmL1 := INT_TO_REAL(iCenterPosition + dataLed.Status.iCuringAreaOffsetL1)/iSlmWidth;
	iFirstCuringBarSlmL1 := REAL_TO_UINT(rFirstCuringBarSlmL1) + 1;

	//To caculate last SLM of the total curing led bar SLMs
	rLastCuringBarSlmL1 := (UINT_TO_REAL(iCenterPosition + dataLed.Status.iCuringAreaOffsetL1 + dataLed.Status.iCuringAreaWidth)/INT_TO_REAL(iSlmWidth));
	pInteger := ADR(rInteger);
	rMantissa := modf(rLastCuringBarSlmL1, pInteger);

	iLastCuringBarSlmL1 := REAL_TO_UINT(rInteger);
	IF rMantissa > 0.0 THEN iLastCuringBarSlmL1 := iLastCuringBarSlmL1 + 1; END_IF
	iLastCuringBarSlmL1 := LIMIT(iFirstCuringBarSlmL1, iLastCuringBarSlmL1, REAL_TO_UINT(iTotalNumSlms/2));

	//Activating curing led bar's SLMs
	FOR iIndexEnableSlm:=iFirstCuringBarSlmL1 TO iLastCuringBarSlmL1 DO
		xCuringLedSlms[iIndexEnableSlm] := TRUE;
	END_FOR

	///////////		L2		///////////
	//To caculate first SLM of the total curing led bar SLMs
	rFirstCuringBarSlmL2 := (UINT_TO_REAL(iCenterPosition + dataLed.Status.iCuringAreaOffsetL2)/INT_TO_REAL(iSlmWidth));
	pInteger := ADR(rInteger);
	rMantissa := modf(rFirstCuringBarSlmL2, pInteger);

	iFirstCuringBarSlmL2 := REAL_TO_UINT(rInteger);
	IF rMantissa > 0.0 THEN iFirstCuringBarSlmL2 := iFirstCuringBarSlmL2 + 1; END_IF
	iFirstCuringBarSlmL2 := LIMIT(iLastCuringBarSlmL1, iFirstCuringBarSlmL2, iTotalNumSlms);

	//To caculate last SLM of the total curing led bar SLMs
	rLastCuringBarSlmL2 := (INT_TO_REAL(iCenterPosition + dataLed.Status.iCuringAreaOffsetL2 + dataLed.Status.iCuringAreaWidth)/INT_TO_REAL(iSlmWidth));
	pInteger := ADR(rInteger);
	rMantissa := modf(rLastCuringBarSlmL2, pInteger);

	iLastCuringBarSlmL2 := REAL_TO_UINT(rInteger);
	IF rMantissa > 0.0 THEN iLastCuringBarSlmL2 := iLastCuringBarSlmL2 + 1; END_IF
	iLastCuringBarSlmL2 := LIMIT(iFirstCuringBarSlmL2, iLastCuringBarSlmL2, iTotalNumSlms);

	FOR iIndexEnableSlm:=iFirstCuringBarSlmL2 TO iLastCuringBarSlmL2 DO
		xCuringLedSlms[iIndexEnableSlm] := TRUE;
	END_FOR

	///////////		To enable lamps stretches		///////////
	iLastLampSLM := 0;
	FOR iIndexEnableLamps:=1 TO iLampsQuantity DO
		iNumLampSLM := dataLed.Lamp[iIndexEnableLamps].Parameters.iNumSLM; //Number of lamp's SLMs

		//Lamp's first SLM of array "xCuringLedSlms" which considers all SLM in the curing led bar
		iFirstLampSLM := iLastLampSLM + 1;
		iLastLampSLM := iLastLampSLM + dataLed.Lamp[iIndexEnableLamps].Parameters.iNumSLM;

		dataLed.Lamp[iIndexEnableLamps].Parameters.xFullActive := TRUE;

		//Calculating slm mirrored to indexSlm. So xCuringLedSlms starts counting from user side to drive side. But lamps are mechanically assemblied in a reverse way, here an image to understand:

		//xCuringLedSlms[x]	  1						  14  15					  28  29					  42  43					  56
		//Lamp's slm index	  14					   1  14					   1  14					   1  14					   1
							//							//							//							//							//
		//FRONT/USER SIDE//	//			1				//			2				//			3				//			4				//		//REAR/WALKWAY SIDE//
							//							//							//							//							//
							//////////////////////////////////////////////////////////////////////////////////////////////////////////////////

		FOR iIndexEnableSlm:=1 TO iNumLampSLM DO
			iMirrorSlm := iLastLampSLM - iIndexEnableSlm + 1;
			dataLed.Lamp[iIndexEnableLamps].Parameters.xSlmEnable[iIndexEnableSlm] := xCuringLedSlms[iMirrorSlm];

			IF (NOT dataLed.Lamp[iIndexEnableLamps].Parameters.xSlmEnable[iIndexEnableSlm]) THEN
				dataLed.Lamp[iIndexEnableLamps].Parameters.xFullActive := FALSE;
			END_IF
		END_FOR
	END_FOR

END_ACTION
```

#### StateManager.st
```iecst
ACTION StateManager:

	xAnyErrorReason.0 := dataChiller.St.Status = CHILLER_FAULT;
	xAnyErrorReason.1 := NitroState = CURINGNITRO_FAULT;
	xAnyErrorReason.2 := errorLampsSLM > 0;
	xAnyErrorReason.3 := errorLampsThermal > 0;
	xAnyError := xAnyErrorReason > 0;

	CASE StatusCtrl OF

		CURINGLED_OFF:
			IF dataLed.Commands.PowerOn THEN
				StatusCtrl := CURINGLED_INIT;
			END_IF

		CURINGLED_INIT:
			IF dataChiller.St.xRunning AND NitroState = CURINGNITRO_READY THEN
				StatusCtrl := CURINGLED_PREPARING;
			END_IF

		CURINGLED_PREPARING:
			IF (dataLed.Status.xCureByStretch AND dataLed.Status.xLampsConfigured) OR NOT dataLed.Status.xCureByStretch THEN
				StatusCtrl := CURINGLED_READY;
			END_IF

		CURINGLED_READY:
			IF dataLed.Commands.RunCuring AND dataLed.Parameters.xEnabled THEN
				StatusCtrl := CURINGLED_EMITTING;
			END_IF

		CURINGLED_EMITTING:
			IF NOT dataLed.Commands.RunCuring OR NOT dataLed.Parameters.xEnabled THEN
				StatusCtrl := CURINGLED_READY;
			END_IF

		CURINGLED_FAULTED:
			IF NOT xAnyError THEN
				StatusCtrl := CURINGLED_INIT;
			END_IF

	END_CASE

	//The enabled lamps with any fault, send the System to fault
	IF xAnyError THEN
		StatusCtrl := CURINGLED_FAULTED;
	END_IF

	IF NOT dataLed.Commands.PowerOn THEN
		StatusCtrl := CURINGLED_OFF;
	END_IF

	dataLed.Status.State:=StatusCtrl;

	//Visu purpose
	dataLed.Status.xEmitting := StatusCtrl = CURINGLED_EMITTING;

END_ACTION
```

### Program Logical/ExtPack/_Cure/CuringLedCtrl/CuringLedSim/CuringLedSim_v1/CuringLedSim (IEC)

#### CuringLedSim.st - Init, cyclic, exit code
```iecst
PROGRAM _INIT
	(* Insert code here *)

END_PROGRAM

PROGRAM _CYCLIC

	dataLed ACCESS ADR (gCuringLed[iIndexCuringLedSim]);

	IF NOT dataLed.Parameters.xInstalled THEN
		iIndexCuringLedSim := iIndexCuringLedSim + 1;
		RETURN;
	END_IF

	iIndexCuringLedSim := iIndexCuringLedSim + 1;

END_PROGRAM
```

- Program Logical/ExtPack/_Cure/CuringLedCtrl/CuringLedSim/CuringLedSim_v1/InitCuringLedSim (IEC) (no source held here)

### Program Logical/ExtPack/_Cure/NIRAdphos/NIRAdphos_v1/NIRAdphosCtrl (IEC)

#### State.st
```iecst
ACTION State:

	xCurrentStateChanged := CurrentState_copy <> CurrentState;
	IF xCurrentStateChanged THEN iStatusChanges := iStatusChanges + 1; END_IF
	CurrentState_copy := CurrentState;

	CASE CurrentState OF
		NIRADPEW_NOT_INITIALIZED:
			ResetSignals;
			IF TRUE THEN
				CurrentState := NIRADPEW_INIT;
			END_IF

		NIRADPEW_COMMS_ERROR:
			IF NOT data.Alarms.xCommsError THEN
				CurrentState := NIRADPEW_NOT_INITIALIZED;
			END_IF

		NIRADPEW_INIT:
			IF data.Signals.In.xSafetyOK THEN
				CurrentState := NIRADPEW_IDLE;
			END_IF

		NIRADPEW_IDLE:
			IF data.Commands.xPrepare THEN
				data.Commands.xPrepare := FALSE;
				CurrentState := NIRADPEW_POWER_ON;
			END_IF
			data.Commands.xStart := FALSE;
			data.Commands.xStop := FALSE;

		NIRADPEW_POWER_ON:
			data.Signals.Out.xPowerOn := TRUE;

			xAllPowered.0 := NOT data.Parameters.Comms.Modules[1].EnableMod OR data.Status.Comms.Modules[1].xPowered;
			xAllPowered.1 := NOT data.Parameters.Comms.Modules[2].EnableMod OR data.Status.Comms.Modules[2].xPowered;
			IF xAllPowered = 16#0003 THEN
				CurrentState := NIRADPEW_POWERED;
			END_IF

		NIRADPEW_POWERED:
			IF data.Status.Comms.xBeltRunning THEN
				CurrentState := NIRADPEW_RUNNING_BELT;
			END_IF

		NIRADPEW_RUNNING_BELT:
			IF data.Signals.In.xReady THEN
				CurrentState := NIRADPEW_READY;
			END_IF
			IF data.Commands.xStop THEN
				data.Commands.xStop := FALSE;
				CurrentState := NIRADPEW_IDLE;
			END_IF

		NIRADPEW_READY:
			IF data.Commands.xStop THEN
				data.Commands.xStop := FALSE;
				CurrentState := NIRADPEW_IDLE;
			ELSIF data.Commands.xStart THEN
				data.Commands.xStart := FALSE;
				CurrentState := NIRADPEW_STARTING;
			END_IF

		NIRADPEW_STARTING:
			IF data.Signals.In.xInProcess THEN
				CurrentState := NIRADPEW_RUNNING;
			END_IF
			IF data.Commands.xStop OR NOT gBelt.states.xRuningBelt THEN
				data.Commands.xStop := FALSE;
				CurrentState := NIRADPEW_IDLE;
			END_IF

		NIRADPEW_RUNNING:
			IF data.Commands.xStop THEN
				data.Commands.xStop := FALSE;
				CurrentState := NIRADPEW_IDLE;
			END_IF

		NIRADPEW_ERROR:
			IF NOT data.Signals.In.xFault THEN
				CurrentState := NIRADPEW_IDLE;
			END_IF

	END_CASE

	IF data.Alarms.xCommsError THEN
		CurrentState := NIRADPEW_COMMS_ERROR;
	END_IF

	IF data.Signals.In.xFault OR NOT data.Parameters.xEnableNir OR data.Parameters.StateMode = PRINTERGEN_ZERO THEN
		CurrentState := NIRADPEW_NOT_INITIALIZED;//NIRADPEW_ERROR
	END_IF

	//Store the history of the status to easy the debug
	IF CurrentState<>StateHistory[0] THEN
		FOR iIndexHistory:=iHistoryLines TO 1 BY -1 DO
			StateHistory[iIndexHistory]:=StateHistory[iIndexHistory-1];
		END_FOR
		StateHistory[0]:=CurrentState;
	END_IF

	data.State := CurrentState;

	//Modules status
	xAnyModuleEnabled := FALSE;
	FOR iIndexModule:=1 TO data.Parameters.iTotalModules DO
		IF data.Parameters.Comms.Modules[iIndexModule].EnableMod THEN
			xAnyModuleEnabled := TRUE;
		END_IF
	END_FOR
	data.Status.xAnyModuleEnabled := xAnyModuleEnabled;

END_ACTION

ACTION ResetSignals:

	data.Signals.Out := SignalsOutReseted;

END_ACTION
```

#### Outputs.st
```iecst
ACTION Outputs:

	//	Digital signals activated in the machine state

	// 100m/min correspond to 10v
	data.Signals.Out.iBeltSpeed:=REAL_TO_INT(data.Parameters.rBeltSpeed * 32766 / 133.0 ); //10V correspond to 32766units
	data.Parameters.Comms.WebWidth := data.Parameters.MediaWidth + MAX(data.Parameters.iExtraDryingWidh, 0);

	iReasonToStop.0 := data.Alarms.xAnyJam;
	iReasonToStop.1 := data.Commands.xExternalSafetyStop;
	iReasonToStop.2 := CurrentState = NIRADPEW_RUNNING AND NOT data.Parameters.xBeltRunning;
	data.Signals.Out.xSafetyStop := iReasonToStop=0; //FALSE to Stop

	iReasonToProcess.0 := CurrentState = NIRADPEW_STARTING;
	iReasonToProcess.1 := CurrentState = NIRADPEW_RUNNING;
	data.Signals.Out.xProcess := iReasonToProcess > 0 AND data.Commands.xMediaInside;

	tonWatchdog.IN:= NOT tonWatchdog.Q;
	tonWatchdog.PT:= T#1s;
	tonWatchdog();
	IF tonWatchdog.Q THEN
		data.Signals.Out.xWatchDog := NOT data.Signals.Out.xWatchDog;
	END_IF

	AdjustMinIntensityDDC;

	ApplyLampsExtendNir1;
	ApplyLampsExtendNir2;

END_ACTION

ACTION AdjustMinIntensityDDC:

	IF NOT data.Status.xEnabledDDC THEN
		RETURN;
	END_IF

	// Protecting for 0 values
	IF data.Status.rPowerSetPoint > 0.1 THEN
		data.Status.iMinPower := MIN(REAL_TO_INT(data.Parameters.DDC.rMinIntensityPercentage / (data.Status.rPowerSetPoint/100.0)), 100);
	ELSE
		data.Status.iMinPower := 0;
	END_IF

END_ACTION

ACTION ApplyLampsExtendNir1:

	IF data.Parameters.DDC.pIntensityNir1 = 0 THEN RETURN; END_IF

	// Assigning data to enable send it to the NIR
	Intensity_Nir1 ACCESS data.Parameters.DDC.pIntensityNir1;

	IF Intensity_Nir1[10] <= 20 THEN
		RETURN;
	END_IF

	IntensityExtend_Nir1 := IntensityReseted_Nir1;

	FOR iIndex_Nir1:=1 TO MIN(THICKENERGY_MAX_LAMPS, data.Parameters.DDC.iLamps) DO
		FOR iIndexExtend_Nir1:= SINT_TO_USINT(MAX(0, USINT_TO_SINT(iIndex_Nir1 - data.Parameters.DDC.iLampsExtend))) TO MIN(THICKENERGY_MAX_LAMPS, iIndex_Nir1 + data.Parameters.DDC.iLampsExtend) DO
			IntensityExtend_Nir1[iIndex_Nir1] := MAX(IntensityExtend_Nir1[iIndex_Nir1], Intensity_Nir1[iIndexExtend_Nir1]);
		END_FOR
	END_FOR

	// Assigning data to the final array
	FOR iIndex_Nir1:=1 TO MIN(THICKENERGY_MAX_LAMPS, data.Parameters.DDC.iLamps) DO
		Intensity_Nir1[iIndex_Nir1] := IntensityExtend_Nir1[iIndex_Nir1];
	END_FOR

END_ACTION

ACTION ApplyLampsExtendNir2:

	IF data.Parameters.DDC.pIntensityNir2 = 0 THEN RETURN; END_IF

	// Assigning data to enable send it to the NIR
	Intensity_Nir2 ACCESS data.Parameters.DDC.pIntensityNir2;

	IF Intensity_Nir2[10] <= 20 THEN
		RETURN;
	END_IF

	IntensityExtend_Nir2 := IntensityReseted_Nir2;

	FOR iIndex_Nir2:=1 TO MIN(THICKENERGY_MAX_LAMPS, data.Parameters.DDC.iLamps) DO
		FOR iIndexExtend_Nir2:= SINT_TO_USINT(MAX(0, USINT_TO_SINT(iIndex_Nir2 - data.Parameters.DDC.iLampsExtend))) TO MIN(THICKENERGY_MAX_LAMPS, iIndex_Nir2 + data.Parameters.DDC.iLampsExtend) DO
			IntensityExtend_Nir2[iIndex_Nir2] := MAX(IntensityExtend_Nir2[iIndex_Nir2], Intensity_Nir2[iIndexExtend_Nir2]);
		END_FOR
	END_FOR

	// Assigning data to the final array
	FOR iIndex_Nir2:=1 TO MIN(THICKENERGY_MAX_LAMPS, data.Parameters.DDC.iLamps) DO
		Intensity_Nir2[iIndex_Nir2] := IntensityExtend_Nir2[iIndex_Nir2];
	END_FOR

END_ACTION
```

#### CommsNir1.st
```iecst
ACTION CommsNir1:

	IF data.Parameters.DDC.pIntensityNir1 = 0 THEN RETURN; END_IF

	// Assigning data to enable send it to the NIR
	Intensity_Nir1 ACCESS data.Parameters.DDC.pIntensityNir1;
	FOR iIndex_Nir1:=0 TO MIN(THICKENERGY_MAX_LAMPS, data.Parameters.DDC.iLamps -1) DO
		iValues_Nir1[iIndex_Nir1] := MAX(Intensity_Nir1[iIndex_Nir1], data.Status.iMinPower);
		data.Status.DDC[1].Intensity[iIndex_Nir1 + 1] := iValues_Nir1[iIndex_Nir1];
	END_FOR

	CASE CommsState_Nir1  OF

		OPCUA_IDLE:

			xAnyCommsError_Nir1 := FALSE;
			IF CurrentState = NIRADPEW_POWER_ON OR CurrentState = NIRADPEW_POWERED OR CurrentState = NIRADPEW_RUNNING_BELT THEN
				CommsState_Nir1 := OPCUA_CONNECTING;
				ExecuteConnect_Nir1 := TRUE;
			END_IF

		OPCUA_CONNECTING: //Connectting

			(* UA_Connect - establish connection to OPC UA Server *)
			SessionConnectInfo_Nir1.SecurityMsgMode := UASecurityMsgMode_None;
			SessionConnectInfo_Nir1.SecurityPolicy := UASecurityPolicy_None;
			SessionConnectInfo_Nir1.TransportProfile := UATP_UATcp;
			SessionConnectInfo_Nir1.UserIdentityToken.UserIdentityTokenType := UAUITT_Anonymous;
			//SessionConnectInfo_Nir1.UserIdentityToken.TokenParam1 := 'PressCore';
			//SessionConnectInfo_Nir1.UserIdentityToken.TokenParam2 := 'h98o76';
			SessionConnectInfo_Nir1.SessionTimeout := T#1m;
			SessionConnectInfo_Nir1.MonitorConnection := T#10s;

			UA_Connect_Nir1(Execute := ExecuteConnect_Nir1,
				ServerEndpointUrl := 'opc.tcp://192.168.125.91:4840',
				SessionConnectInfo := SessionConnectInfo_Nir1,
				Timeout := T#10s
			);

			IF NOT UA_Connect_Nir1.Busy THEN
				ExecuteConnect_Nir1 := FALSE;
				IF UA_Connect_Nir1.Done THEN
					ConnectionHdl_Nir1 := UA_Connect_Nir1.ConnectionHdl;
					////// NEXT
					CommsState_Nir1 := OPCUA_GETTING_NAMESPACE;
					ExecuteGetnamespaceindex_Nir1 := TRUE;
					iTimes_Nir1 := 0;
				END_IF
				IF UA_Connect_Nir1.Error THEN
					ConnectionHdl_Nir1 := 0;
					xAnyCommsError_Nir1 := TRUE;
					ExecuteNodeReleaseHandle_Nir1 := TRUE;
					CommsState_Nir1 := OPCUA_RELEASINSG_HANDLE;
				END_IF
				UA_Connect_Nir1(Execute := ExecuteConnect_Nir1);
			END_IF

			iTimes_Nir1 := iTimes_Nir1 + 1;

		OPCUA_GETTING_NAMESPACE:

			(* UA_GetNamespaceIndex - read index of required namespace for PVs *)
			UA_GetNamespaceIndex_Nir1(Execute := ExecuteGetnamespaceindex_Nir1,
				ConnectionHdl := ConnectionHdl_Nir1,
				NamespaceUri := 'http://RecData',
				Timeout := T#5s
			);

			IF NOT UA_GetNamespaceIndex_Nir1.Busy THEN
				ExecuteGetnamespaceindex_Nir1 := FALSE;
				IF UA_GetNamespaceIndex_Nir1.Done THEN
					NamespaceIndex_Nir1 := UA_GetNamespaceIndex_Nir1.NamespaceIndex;
					////// NEXT
					CommsState_Nir1 := OPCUA_GETTING_HANDLE;
					ExecuteMethodGetHandle_Nir1 := TRUE;
					iTimes_Nir1 := 0;
				END_IF
				IF UA_GetNamespaceIndex_Nir1.Error THEN
					NamespaceIndex_Nir1 := 0;
					xAnyCommsError_Nir1 := TRUE;
					ExecuteNodeReleaseHandle_Nir1 := TRUE;
					CommsState_Nir1 := OPCUA_RELEASINSG_HANDLE;
				END_IF
				UA_GetNamespaceIndex_Nir1(Execute := ExecuteGetnamespaceindex_Nir1);
			END_IF

			iTimes_Nir1 := iTimes_Nir1 + 1;

		OPCUA_GETTING_HANDLE:

			(* UA_NodeGetHandle - get a handle for required methode *)
			ObjectNodeID_Nir1.NamespaceIndex := NamespaceIndex_Nir1;
			ObjectNodeID_Nir1.Identifier := '27';
			ObjectNodeID_Nir1.IdentifierType := UAIdentifierType_Numeric;

			UA_NodeGetHandle_Nir1(Execute := ExecuteMethodGetHandle_Nir1,
				ConnectionHdl := ConnectionHdl_Nir1,
				NodeID := ObjectNodeID_Nir1,
				Timeout := T#10s
			);

			IF NOT UA_NodeGetHandle_Nir1.Busy THEN
				ExecuteMethodGetHandle_Nir1 := FALSE;
				IF UA_NodeGetHandle_Nir1.Done THEN
					NodeHdl_Nir1 := UA_NodeGetHandle_Nir1.NodeHdl;
					////// NEXT
					CommsState_Nir1 := OPCUA_EXECUTING;
					iTimes_Nir1 := 0;
					// READY TO COMMUNICATE
				END_IF
				IF UA_NodeGetHandle_Nir1.Error THEN
					NodeHdl_Nir1 := 0;
					xAnyCommsError_Nir1 := TRUE;
					ExecuteNodeReleaseHandle_Nir1 := TRUE;
					CommsState_Nir1 := OPCUA_RELEASINSG_HANDLE;
				END_IF
				UA_NodeGetHandle_Nir1(Execute := ExecuteMethodGetHandle_Nir1);
			END_IF

			iTimes_Nir1 := iTimes_Nir1 + 1;

		OPCUA_EXECUTING:

			(* UA_Write - call methode *)
			IndexRange_Nir1.StartIndex := 0;
			IndexRange_Nir1.EndIndex := 0;
			NodeAddInfo_Nir1.AttributeId := UAAI_Value;
			NodeAddInfo_Nir1.IndexRangeCount := 0;
			NodeAddInfo_Nir1.IndexRange[0] := IndexRange_Nir1;

			UA_Write_Nir1(Execute := ExecuteMethodCall_Nir1,
				ConnectionHdl := ConnectionHdl_Nir1,
				NodeHdl := NodeHdl_Nir1,
				NodeAddInfo := NodeAddInfo_Nir1,
				Timeout := T#10s,
				Variable := '::NIRAdphos:iValues_Nir1'
			);

			IF NOT UA_Write_Nir1.Busy THEN
				ExecuteMethodCall_Nir1 := FALSE;

				IF UA_Write_Nir1.Done THEN
					iGoodComms_Nir1 := iGoodComms_Nir1 + 1;
					iPartialGoodTimes_Nir1 := iPartialGoodTimes_Nir1 + 1;
				END_IF

				IF UA_Write_Nir1.Error THEN
					xAnyCommsError_Nir1 := TRUE;
					ExecuteNodeReleaseHandle_Nir1 := TRUE;
					CommsState_Nir1 := OPCUA_RELEASINSG_HANDLE;
				END_IF

				// Exiting from Executing when no communicating
				IF CurrentState = NIRADPEW_IDLE THEN
					ExecuteNodeReleaseHandle_Nir1 := TRUE;
					CommsState_Nir1 := OPCUA_RELEASINSG_HANDLE;
					iTimes_Nir1 := 0;
				END_IF
				UA_Write_Nir1(Execute := ExecuteMethodCall_Nir1, Variable := '::NIRAdphos:iValues_Nir1');

			END_IF

			tonNextComms_Nir1.IN := NOT ExecuteMethodCall_Nir1;
			IF tonNextComms_Nir1.PT = 0 THEN
				tonNextComms_Nir1.PT := T#20ms;
			END_IF
			tonNextComms_Nir1();
			IF tonNextComms_Nir1.Q THEN
				ExecuteMethodCall_Nir1 := TRUE;
				// Update values in simulation just for comms
				IF gDryer.St.HwData.Family = FAMILY_BRAUTOMATIONRUNTIME THEN
					UpdateSimDataForMediaNir1;
				END_IF
			END_IF

			iTimes_Nir1 := iTimes_Nir1 + 1;

		OPCUA_PAUSED:

		OPCUA_RELEASINSG_HANDLE:

			UA_NodeReleaseHandle_Nir1(Execute := ExecuteNodeReleaseHandle_Nir1,
				ConnectionHdl := ConnectionHdl_Nir1,
				NodeHdl := NodeHdl_Nir1,
				Timeout := T#10s
			);

			IF NOT UA_NodeReleaseHandle_Nir1.Busy THEN
				ExecuteNodeReleaseHandle_Nir1 := FALSE;

				IF UA_NodeReleaseHandle_Nir1.Done THEN
					////// NEXT
					NodeHdl_Nir1 := 0;
					ExecuteDisconnect_Nir1 := TRUE;
					CommsState_Nir1 := OPCUA_DISCONNECTING;
					iTimes_Nir1 := 0;
				END_IF
				IF UA_NodeReleaseHandle_Nir1.Error THEN
					NodeHdl_Nir1 := 0;
					xAnyCommsError_Nir1 := TRUE;
					ExecuteDisconnect_Nir1 := TRUE;
					CommsState_Nir1 := OPCUA_DISCONNECTING;
				END_IF

				UA_NodeReleaseHandle_Nir1(Execute := ExecuteNodeReleaseHandle_Nir1);
			END_IF

			iTimes_Nir1 := iTimes_Nir1 + 1;

		OPCUA_DISCONNECTING:

			UA_Disconnect_Nir1(Execute := ExecuteDisconnect_Nir1,
				ConnectionHdl := ConnectionHdl_Nir1,
				Timeout := T#10s
			);

			IF NOT UA_Disconnect_Nir1.Busy THEN
				ExecuteDisconnect_Nir1 := FALSE;

				IF UA_Disconnect_Nir1.Done THEN
					////// NEXT
					ConnectionHdl_Nir1 := 0;
					// If arriving here after any error, go to error before going to Idle
					IF xAnyCommsError_Nir1 THEN
						CommsState_Nir1 := OPCUA_FAULTED;
					ELSE
						CommsState_Nir1 := OPCUA_IDLE;
					END_IF
				END_IF
				IF UA_Disconnect_Nir1.Error THEN
					ConnectionHdl_Nir1 := 0;
					CommsState_Nir1 := OPCUA_FAULTED;
				END_IF

				UA_Disconnect_Nir1(Execute := ExecuteDisconnect_Nir1);
			END_IF

		OPCUA_FAULTED:

			tonWaitExitFault_Nir1.IN := TRUE;
			tonWaitExitFault_Nir1.PT := T#2s;
			tonWaitExitFault_Nir1();
			IF tonWaitExitFault_Nir1.Q THEN
				tonWaitExitFault_Nir1(IN:=FALSE); //This is neccessary to allow the timer working in the second time entering here
				CommsState_Nir1 := OPCUA_IDLE;
			END_IF

	END_CASE

	// If an error is detected, raise the alarm. Wait to free resouces before allow reseting alarm
	IF xAnyCommsError_Nir1 THEN
		data.Alarms.xOpcUaWriteError[iIndexConstant_Nir1] := TRUE;
	END_IF

	// Update ratio calculation
	IF tonCalculateUpdate_Nir1.Q THEN
		IF iPartialGoodTimes_Nir1 > 0 THEN
			rUpdateRatio_Nir1 := 1000 * 10.0 / UINT_TO_REAL(iPartialGoodTimes_Nir1);
		ELSE
			rUpdateRatio_Nir1 := 0;
		END_IF
		iPartialGoodTimes_Nir1 := 0;
	END_IF
	tonCalculateUpdate_Nir1.IN := NOT tonCalculateUpdate_Nir1.Q;
	tonCalculateUpdate_Nir1.PT := t#10s;
	tonCalculateUpdate_Nir1();

	// Manage History of status
	IF CommsState_Nir1<>StateHistory_Nir1[0] THEN
		FOR iIndexHistory:=iHistoryLines TO 1 BY -1 DO
			StateHistory_Nir1[iIndexHistory] := StateHistory_Nir1[iIndexHistory-1];
		END_FOR
		StateHistory_Nir1[0]:=CommsState_Nir1;
	END_IF

END_ACTION

ACTION InitialDataForMediaNir1:

	FOR iIndexValue_Nir1 := 0 TO 47 DO
		iValues_Nir1[iIndexValue_Nir1] := iIndexValue_Nir1;
	END_FOR

END_ACTION

ACTION UpdateSimDataForMediaNir1:

	FOR iIndexValue_Nir1 := 0 TO 47 DO
		iValues_Nir1[iIndexValue_Nir1] := iValues_Nir1[iIndexValue_Nir1] + 1;
		IF iValues_Nir1[iIndexValue_Nir1] > 100 THEN
			iValues_Nir1[iIndexValue_Nir1] := 0;
		END_IF
	END_FOR

END_ACTION

ACTION PreparingMethodCommsNir1:

END_ACTION
```

#### CommsNir2.st
```iecst
ACTION CommsNir2:

	IF data.Parameters.DDC.pIntensityNir2 = 0 THEN RETURN; END_IF

	// Assigning data to enable send it to the NIR
	Intensity_Nir2 ACCESS data.Parameters.DDC.pIntensityNir2;
	FOR iIndex_Nir2:=0 TO MIN(THICKENERGY_MAX_LAMPS, data.Parameters.DDC.iLamps -1) DO
		iValues_Nir2[iIndex_Nir2] := MAX(Intensity_Nir2[iIndex_Nir2], data.Status.iMinPower);
		data.Status.DDC[2].Intensity[iIndex_Nir2 + 1] := iValues_Nir2[iIndex_Nir2];
	END_FOR

	CASE CommsState_Nir2  OF

		OPCUA_IDLE:

			xAnyCommsError_Nir2 := FALSE;
			IF CurrentState = NIRADPEW_POWER_ON OR CurrentState = NIRADPEW_POWERED OR CurrentState = NIRADPEW_RUNNING_BELT THEN
				CommsState_Nir2 := OPCUA_CONNECTING;
				ExecuteConnect_Nir2 := TRUE;
			END_IF

		OPCUA_CONNECTING: //Connectting

			(* UA_Connect - establish connection to OPC UA Server *)
			SessionConnectInfo_Nir2.SecurityMsgMode := UASecurityMsgMode_None;
			SessionConnectInfo_Nir2.SecurityPolicy := UASecurityPolicy_None;
			SessionConnectInfo_Nir2.TransportProfile := UATP_UATcp;
			SessionConnectInfo_Nir2.UserIdentityToken.UserIdentityTokenType := UAUITT_Anonymous;
			//SessionConnectInfo_Nir2.UserIdentityToken.TokenParam1 := 'PressCore';
			//SessionConnectInfo_Nir2.UserIdentityToken.TokenParam2 := 'h98o76';
			SessionConnectInfo_Nir2.SessionTimeout := T#1m;
			SessionConnectInfo_Nir2.MonitorConnection := T#10s;

			UA_Connect_Nir2(Execute := ExecuteConnect_Nir2,
				ServerEndpointUrl := 'opc.tcp://192.168.125.92:4840',
				SessionConnectInfo := SessionConnectInfo_Nir2,
				Timeout := T#10s
			);

			IF NOT UA_Connect_Nir2.Busy THEN
				ExecuteConnect_Nir2 := FALSE;
				IF UA_Connect_Nir2.Done THEN
					ConnectionHdl_Nir2 := UA_Connect_Nir2.ConnectionHdl;
					////// NEXT
					CommsState_Nir2 := OPCUA_GETTING_NAMESPACE;
					ExecuteGetnamespaceindex_Nir2 := TRUE;
					iTimes_Nir2 := 0;
				END_IF
				IF UA_Connect_Nir2.Error THEN
					ConnectionHdl_Nir2 := 0;
					xAnyCommsError_Nir2 := TRUE;
					ExecuteNodeReleaseHandle_Nir2 := TRUE;
					CommsState_Nir2 := OPCUA_RELEASINSG_HANDLE;
				END_IF
				UA_Connect_Nir2(Execute := ExecuteConnect_Nir2);
			END_IF

			iTimes_Nir2 := iTimes_Nir2 + 1;

		OPCUA_GETTING_NAMESPACE:

			(* UA_GetNamespaceIndex - read index of required namespace for PVs *)
			UA_GetNamespaceIndex_Nir2(Execute := ExecuteGetnamespaceindex_Nir2,
				ConnectionHdl := ConnectionHdl_Nir2,
				NamespaceUri := 'http://RecData',
				Timeout := T#5s
			);

			IF NOT UA_GetNamespaceIndex_Nir2.Busy THEN
				ExecuteGetnamespaceindex_Nir2 := FALSE;
				IF UA_GetNamespaceIndex_Nir2.Done THEN
					NamespaceIndex_Nir2 := UA_GetNamespaceIndex_Nir2.NamespaceIndex;
					////// NEXT
					CommsState_Nir2 := OPCUA_GETTING_HANDLE;
					ExecuteMethodGetHandle_Nir2 := TRUE;
					iTimes_Nir2 := 0;
				END_IF
				IF UA_GetNamespaceIndex_Nir2.Error THEN
					NamespaceIndex_Nir2 := 0;
					xAnyCommsError_Nir2 := TRUE;
					ExecuteNodeReleaseHandle_Nir2 := TRUE;
					CommsState_Nir2 := OPCUA_RELEASINSG_HANDLE;
				END_IF
				UA_GetNamespaceIndex_Nir2(Execute := ExecuteGetnamespaceindex_Nir2);
			END_IF

			iTimes_Nir2 := iTimes_Nir2 + 1;

		OPCUA_GETTING_HANDLE:

			(* UA_NodeGetHandle - get a handle for required methode *)
			ObjectNodeID_Nir2.NamespaceIndex := NamespaceIndex_Nir2;
			ObjectNodeID_Nir2.Identifier := '6';
			ObjectNodeID_Nir2.IdentifierType := UAIdentifierType_Numeric;

			UA_NodeGetHandle_Nir2(Execute := ExecuteMethodGetHandle_Nir2,
				ConnectionHdl := ConnectionHdl_Nir2,
				NodeID := ObjectNodeID_Nir2,
				Timeout := T#10s
			);

			IF NOT UA_NodeGetHandle_Nir2.Busy THEN
				ExecuteMethodGetHandle_Nir2 := FALSE;
				IF UA_NodeGetHandle_Nir2.Done THEN
					NodeHdl_Nir2 := UA_NodeGetHandle_Nir2.NodeHdl;
					////// NEXT
					CommsState_Nir2 := OPCUA_EXECUTING;
					iTimes_Nir2 := 0;
					// READY TO COMMUNICATE
				END_IF
				IF UA_NodeGetHandle_Nir2.Error THEN
					NodeHdl_Nir2 := 0;
					xAnyCommsError_Nir2 := TRUE;
					ExecuteNodeReleaseHandle_Nir2 := TRUE;
					CommsState_Nir2 := OPCUA_RELEASINSG_HANDLE;
				END_IF
				UA_NodeGetHandle_Nir2(Execute := ExecuteMethodGetHandle_Nir2);
			END_IF

			iTimes_Nir2 := iTimes_Nir2 + 1;

		OPCUA_EXECUTING:

			(* UA_Write - call methode *)
			IndexRange_Nir2.StartIndex := 0;
			IndexRange_Nir2.EndIndex := 0;
			NodeAddInfo_Nir2.AttributeId := UAAI_Value;
			NodeAddInfo_Nir2.IndexRangeCount := 0;
			NodeAddInfo_Nir2.IndexRange[0] := IndexRange_Nir2;

			UA_Write_Nir2(Execute := ExecuteMethodCall_Nir2,
				ConnectionHdl := ConnectionHdl_Nir2,
				NodeHdl := NodeHdl_Nir2,
				NodeAddInfo := NodeAddInfo_Nir2,
				Timeout := T#10s,
				Variable := '::NIRAdphos:iValues_Nir2'
			);

			IF NOT UA_Write_Nir2.Busy THEN
				ExecuteMethodCall_Nir2 := FALSE;

				IF UA_Write_Nir2.Done THEN
					iGoodComms_Nir2 := iGoodComms_Nir2 + 1;
					iPartialGoodTimes_Nir2 := iPartialGoodTimes_Nir2 + 1;
				END_IF

				IF UA_Write_Nir2.Error THEN
					xAnyCommsError_Nir2 := TRUE;
					ExecuteNodeReleaseHandle_Nir2 := TRUE;
					CommsState_Nir2 := OPCUA_RELEASINSG_HANDLE;
				END_IF

				// Exiting from Executing when no communicating
				IF CurrentState = NIRADPEW_IDLE THEN
					ExecuteNodeReleaseHandle_Nir2 := TRUE;
					CommsState_Nir2 := OPCUA_RELEASINSG_HANDLE;
					iTimes_Nir2 := 0;
				END_IF
				UA_Write_Nir2(Execute := ExecuteMethodCall_Nir2, Variable := '::NIRAdphos:iValues_Nir2');

			END_IF

			tonNextComms_Nir2.IN := NOT ExecuteMethodCall_Nir2;
			IF tonNextComms_Nir2.PT = 0 THEN
				tonNextComms_Nir2.PT := T#20ms;
			END_IF
			tonNextComms_Nir2();
			IF tonNextComms_Nir2.Q THEN
				ExecuteMethodCall_Nir2 := TRUE;
				// Update values in simulation just for comms
				IF gDryer.St.HwData.Family = FAMILY_BRAUTOMATIONRUNTIME THEN
					UpdateSimDataForMediaNir2;
				END_IF
			END_IF

			iTimes_Nir2 := iTimes_Nir2 + 1;

		OPCUA_PAUSED:

		OPCUA_RELEASINSG_HANDLE:

			UA_NodeReleaseHandle_Nir2(Execute := ExecuteNodeReleaseHandle_Nir2,
				ConnectionHdl := ConnectionHdl_Nir2,
				NodeHdl := NodeHdl_Nir2,
				Timeout := T#10s
			);

			IF NOT UA_NodeReleaseHandle_Nir2.Busy THEN
				ExecuteNodeReleaseHandle_Nir2 := FALSE;

				IF UA_NodeReleaseHandle_Nir2.Done THEN
					////// NEXT
					NodeHdl_Nir2 := 0;
					ExecuteDisconnect_Nir2 := TRUE;
					CommsState_Nir2 := OPCUA_DISCONNECTING;
					iTimes_Nir2 := 0;
				END_IF
				IF UA_NodeReleaseHandle_Nir2.Error THEN
					NodeHdl_Nir2 := 0;
					xAnyCommsError_Nir2 := TRUE;
					ExecuteDisconnect_Nir2 := TRUE;
					CommsState_Nir2 := OPCUA_DISCONNECTING;
				END_IF

				UA_NodeReleaseHandle_Nir2(Execute := ExecuteNodeReleaseHandle_Nir2);
			END_IF

			iTimes_Nir2 := iTimes_Nir2 + 1;

		OPCUA_DISCONNECTING:

			UA_Disconnect_Nir2(Execute := ExecuteDisconnect_Nir2,
				ConnectionHdl := ConnectionHdl_Nir2,
				Timeout := T#10s
			);

			IF NOT UA_Disconnect_Nir2.Busy THEN
				ExecuteDisconnect_Nir2 := FALSE;

				IF UA_Disconnect_Nir2.Done THEN
					////// NEXT
					ConnectionHdl_Nir2 := 0;
					// If arriving here after any error, go to error before going to Idle
					IF xAnyCommsError_Nir2 THEN
						CommsState_Nir2 := OPCUA_FAULTED;
					ELSE
						CommsState_Nir2 := OPCUA_IDLE;
					END_IF
				END_IF
				IF UA_Disconnect_Nir2.Error THEN
					ConnectionHdl_Nir2 := 0;
					CommsState_Nir2 := OPCUA_FAULTED;
				END_IF

				UA_Disconnect_Nir2(Execute := ExecuteDisconnect_Nir2);
			END_IF

		OPCUA_FAULTED:

			tonWaitExitFault_Nir2.IN := TRUE;
			tonWaitExitFault_Nir2.PT := T#2s;
			tonWaitExitFault_Nir2();
			IF tonWaitExitFault_Nir2.Q THEN
				tonWaitExitFault_Nir2(IN:=FALSE); //This is neccessary to allow the timer working in the second time entering here
				CommsState_Nir2 := OPCUA_IDLE;
			END_IF

	END_CASE

	// If an error is detected, raise the alarm. Wait to free resouces before allow reseting alarm
	IF xAnyCommsError_Nir2 THEN
		data.Alarms.xOpcUaWriteError[iIndexConstant_Nir2] := TRUE;
	END_IF

	// Update ratio calculation
	IF tonCalculateUpdate_Nir2.Q THEN
		IF iPartialGoodTimes_Nir2 > 0 THEN
			rUpdateRatio_Nir2 := 1000 * 10.0 / UINT_TO_REAL(iPartialGoodTimes_Nir2);
		ELSE
			rUpdateRatio_Nir2 := 0;
		END_IF
		iPartialGoodTimes_Nir2 := 0;
	END_IF
	tonCalculateUpdate_Nir2.IN := NOT tonCalculateUpdate_Nir2.Q;
	tonCalculateUpdate_Nir2.PT := t#10s;
	tonCalculateUpdate_Nir2();

	// Manage History of status
	IF CommsState_Nir2<>StateHistory_Nir2[0] THEN
		FOR iIndexHistory:=iHistoryLines TO 1 BY -1 DO
			StateHistory_Nir2[iIndexHistory] := StateHistory_Nir2[iIndexHistory-1];
		END_FOR
		StateHistory_Nir2[0]:=CommsState_Nir2;
	END_IF

END_ACTION

ACTION InitialDataForMediaNir2:

	FOR iIndexValue_Nir2 := 0 TO 47 DO
		iValues_Nir2[iIndexValue_Nir2] := iIndexValue_Nir2;
	END_FOR

END_ACTION

ACTION UpdateSimDataForMediaNir2:

	FOR iIndexValue_Nir2 := 0 TO 47 DO
		iValues_Nir2[iIndexValue_Nir2] := iValues_Nir2[iIndexValue_Nir2] + 1;
		IF iValues_Nir2[iIndexValue_Nir2] > 100 THEN
			iValues_Nir2[iIndexValue_Nir2] := 0;
		END_IF
	END_FOR

END_ACTION

ACTION PreparingMethodCommsNir2:

END_ACTION
```

#### EventLog.st
```iecst
ACTION LogStopAlarm:

//	iReasonStop.0 := data.Alarms.xCommsError;
//	iReasonStop.1 := data.Alarms.xMaxSurfaceTempModule[1];
//	iReasonStop.2 := data.Alarms.xMaxSurfaceTempModule[2];
//	iReasonStop.3 := data.Alarms.xFault;
//	iReasonStop.4 := data.Alarms.xAnyJam;
//	iReasonStop.5 := data.Alarms.xOpcUaWriteError[1] AND data.Status.xEnabledDDC;
//	iReasonStop.6 := data.Alarms.xOpcUaWriteError[2] AND data.Status.xEnabledDDC;

	stEventLog.Source := ELOG_TYPE_NIR;
	stEventLog.Severity:= ELOG_SEVERITY_ERROR;
	stEventLog.Facility:= 0;
	stEventLog.ErrorCode:=0;

	stEventLog.Text := 'NIR.LogStopAlarm';

	IF 		iReasonStop.0 THEN stEventLog.Text := 'NirStop. xCommsError';
	ELSIF 	iReasonStop.1 THEN stEventLog.Text := 'NirStop. xMaxSurfaceTempModule[1]';
	ELSIF 	iReasonStop.2 THEN stEventLog.Text := 'NirStop. xMaxSurfaceTempModule[2]';
	ELSIF 	iReasonStop.3 THEN stEventLog.Text := 'NirStop. xFault';
	ELSIF 	iReasonStop.4 THEN stEventLog.Text := 'NirStop. xAnyJam';
	ELSIF 	iReasonStop.5 THEN stEventLog.Text := 'NirStop. xOpcUaWriteError[1]';
	ELSIF 	iReasonStop.6 THEN stEventLog.Text := 'NirStop. xOpcUaWriteError[2]';
	END_IF

	gEventLogLoader(EventData := ADR(stEventLog));

END_ACTION

ACTION LogCriticalAlarm:

//	iReasonCritical.0 := data.Status.Comms.Modules[1].error;
//	iReasonCritical.1 := data.Status.Comms.Modules[2].error;
//	iReasonCritical.2 := data.Alarms.xSafetyError;

	stEventLog.Source := ELOG_TYPE_NIR;
	stEventLog.Severity:= ELOG_SEVERITY_ERROR;
	stEventLog.Facility:= 0;
	stEventLog.ErrorCode:=0;

	stEventLog.Text := 'NIR.LogCriticalAlarm';

	IF 		iReasonCritical.0 THEN stEventLog.Text := 'NirCrit. Modules[1].error';
	ELSIF 	iReasonCritical.1 THEN stEventLog.Text := 'NirCrit. Modules[2].error';
	ELSIF 	iReasonCritical.2 THEN stEventLog.Text := 'NirCrit. xSafetyError';
	END_IF

	gEventLogLoader(EventData := ADR(stEventLog));

END_ACTION
```

#### NIRAdphosCtrl.var - Local variables
```iecst
VAR
	data : REFERENCE TO NIRAdphos;
	CurrentState : NIRAdphos_State := NIRADPEW_NOT_INITIALIZED;
	CurrentState_copy : NIRAdphos_State := NIRADPEW_NOT_INITIALIZED;
	resetedAlarms : NIRAdphos_Alarms;
	resetedAlarmsSummary : stEFI_AlarmSummary;
	xCurrentStateChanged : BOOL;
	iStatusChanges : UINT;
	SignalsOutReseted : NIRAdphos_SignalsOut;
	xAllPowered : UINT;
	iIndexModule : USINT;
	iReasonStop : UINT;
	iReasonCritical : UINT;
	iAnyAlarm : UINT;
	iAnyWarning : UINT;
	stEventLog : EventLog_typ;
	reasonSound : UINT;
	arFault : AutoResetSound;
	arSafety : AutoResetSound;
	arSurfaceTemp1 : AutoResetSound;
	arSurfaceTemp2 : AutoResetSound;
	tonWatchdog : TON;
	arSurfaceTempSensorError1 : AutoResetSound;
	arSurfaceTempSensorError2 : AutoResetSound;
	arAnyBlockedFan : AutoResetSound;
	arAnyJam : AutoResetSound;
	xAnyBlockedFan : BOOL;
	xAnyJam : BOOL;
	iIndexFan : USINT;
	iReasonToProcess : USINT;
	iReasonToStop : USINT;
	xAnyModuleEnabled : BOOL;
END_VAR
VAR CONSTANT
	iHistoryLines : USINT := 25;
END_VAR
VAR
	StateHistory : ARRAY[0..iHistoryLines] OF NIRAdphos_State;
	iIndexHistory : USINT;
END_VAR
```

- NIRAdphosStates.graphml - Photocell states ctrl (not shown)

### Program Logical/ExtPack/_Cure/NIRAdphos/NirAdphosSim/NirAdphosSim_v1/NirAdphosSim (IEC)

#### Comms.st
```iecst
ACTION EndComms:

	IF tonCommand.Q	THEN
		dataNir.Status.CommsStatus := ARCLG_IDLE;
		dataNir.Commands.InternalComms := CommsCmdReseted;
	END_IF

END_ACTION
```

#### NirAdphosSim.st
```iecst
PROGRAM _INIT

	dataNir ACCESS ADR(gNirAdphos);

	dataNir.Signals.In.xSafetyOK := TRUE;

	dataNir.Parameters.iTotalModules:= 2;

	dataNir.Parameters.Comms.AdjPos := 0;
	dataNir.Parameters.Comms.Pstart := 0;
	dataNir.Parameters.Comms.Pend := 100;
	dataNir.Parameters.Comms.Vstart := 0;
	dataNir.Parameters.Comms.Vend := 100;

	dataNir.Parameters.Comms.Modules[1].EnableMod := TRUE;
	dataNir.Parameters.Comms.Modules[1].Adjust := 0;
	dataNir.Parameters.Comms.Modules[2].EnableMod := TRUE;
	dataNir.Parameters.Comms.Modules[2].Adjust := 0;

	dataNir.Status.xCommsOK := TRUE;

	iMaxTemperature := 500;
	iMinTemperature := 250;

END_PROGRAM

PROGRAM _CYCLIC
	(* Insert code here *)
	dataNir ACCESS ADR(gNirAdphos);
	SimNirAdphos ACCESS ADR(gSimNirAdphos);

	tonReady.IN := dataNir.State = NIRADPEW_RUNNING_BELT;
	tonReady.PT:= T#1s;
	tonReady();
	IF tonReady.Q THEN
		dataNir.Signals.In.xReady := TRUE;
	END_IF

	tonDry.IN:= dataNir.Signals.Out.xProcess;
	tonDry.PT:= T#1s;
	tonDry();
	IF tonDry.Q THEN
		dataNir.Signals.In.xInProcess := TRUE;
	END_IF

	FOR iIndexModule := 1 TO dataNir.Parameters.iTotalModules DO
		IF dataNir.Signals.Out.xPowerOn THEN

			rModulePowerSetPoint := dataNir.Status.rPowerSetPoint * (1 + INT_TO_REAL(dataNir.Parameters.Comms.Modules[iIndexModule].Adjust)/100);
			rModulePowerSetPoint := MIN(rModulePowerSetPoint, 100);

			IF dataNir.Parameters.Comms.Modules[iIndexModule].EnableMod AND rModulePower[iIndexModule]  < rModulePowerSetPoint THEN
				rModulePower[iIndexModule] := MIN(rModulePower[iIndexModule] + POWER_VARIATION, rModulePowerSetPoint);
			ELSE
				rModulePower[iIndexModule] := MAX(rModulePower[iIndexModule] - POWER_VARIATION, rModulePowerSetPoint);
			END_IF

			IF dataNir.Parameters.Comms.Modules[iIndexModule].EnableMod AND dataNir.Signals.In.iSurfaceTempModuleRaw[iIndexModule]  < iMaxTemperature THEN
				IF tonDelayTemp.Q THEN dataNir.Signals.In.iSurfaceTempModuleRaw[iIndexModule] := MIN(dataNir.Signals.In.iSurfaceTempModuleRaw[iIndexModule] + 1, iMaxTemperature); END_IF
			ELSE
				IF tonDelayTemp.Q THEN dataNir.Signals.In.iSurfaceTempModuleRaw[iIndexModule] := MAX(dataNir.Signals.In.iSurfaceTempModuleRaw[iIndexModule] - 1, iMinTemperature); END_IF
			END_IF

			//NIR Module Status
			IF dataNir.Parameters.Comms.Modules[iIndexModule].EnableMod THEN
				IF dataNir.Signals.Out.xProcess THEN
					dataNir.Status.Comms.Modules[iIndexModule].iNirStatus := 4;
				ELSE
					dataNir.Status.Comms.Modules[iIndexModule].iNirStatus := 2;
				END_IF
			ELSE
				dataNir.Status.Comms.Modules[iIndexModule].iNirStatus := 0;
			END_IF
		ELSE
			rModulePower[iIndexModule] := MAX(rModulePower[iIndexModule] - POWER_VARIATION, 0);
			IF tonDelayTemp.Q THEN dataNir.Signals.In.iSurfaceTempModuleRaw[iIndexModule] := MAX(dataNir.Signals.In.iSurfaceTempModuleRaw[iIndexModule] - 1, iMinTemperature); END_IF

			dataNir.Status.Comms.Modules[iIndexModule].iNirStatus := 0;
		END_IF

		dataNir.Status.Comms.Modules[iIndexModule].Power := REAL_TO_INT(rModulePower[iIndexModule]);
		dataNir.Status.Comms.Modules[iIndexModule].xPowered := dataNir.Signals.Out.xPowerOn AND dataNir.Parameters.Comms.Modules[iIndexModule].EnableMod;
	END_FOR;

	tonDelayTemp.IN := NOT tonDelayTemp.Q;
	IF dataNir.Signals.Out.xProcess THEN
		tonDelayTemp.PT := t#200ms;
	ELSIF dataNir.Signals.Out.xPowerOn THEN
			tonDelayTemp.PT := t#1s;
	ELSE
		tonDelayTemp.PT := t#2s;
	END_IF
	tonDelayTemp();

	tonPowerOn.IN:= dataNir.Signals.Out.xPowerOn;
	tonPowerOn.PT:= T#1s;
	tonPowerOn();
	IF tonPowerOn.Q THEN
		//dataNir.Status.Comms.xPowered := TRUE;
	END_IF

	iReasonBeltRunning.0 := dataNir.State = NIRADPEW_POWERED;
	iReasonBeltRunning.1 := dataNir.State = NIRADPEW_RUNNING_BELT;
	iReasonBeltRunning.2 := dataNir.State = NIRADPEW_READY;
	iReasonBeltRunning.3 := dataNir.State = NIRADPEW_STARTING;
	iReasonBeltRunning.4 := dataNir.State = NIRADPEW_RUNNING;

	IF iReasonBeltRunning > 0 THEN
		dataNir.Status.Comms.Speed := SimNirAdphos.Parameters.CurrentSpeed;
	ELSE
		dataNir.Status.Comms.Speed := 0;
	END_IF

	IF EDGEPOS(dataNir.State = NIRADPEW_IDLE) THEN
		dataNir.Signals.In.xFault := FALSE;
		dataNir.Signals.In.xInProcess := FALSE;
		dataNir.Signals.In.xReady := FALSE;
		dataNir.Signals.In.xSafetyOK := TRUE;
		dataNir.Status.Comms := StatusCommsReseted;
	END_IF

	// It is working because comms are executed after AlarmSummary
	dataNir.Alarms.xOpcUaWriteError[1] := FALSE;
	dataNir.Alarms.xOpcUaWriteError[2] := FALSE;

END_PROGRAM
```

### Chiller.typ
```iecst
TYPE
	ChillerSystemType_enum :
		(
		CHILLERSYS_UNDEFINED,
		CHILLERSYS_DIRECT,
		CHILLERSYS_WATERMANIFOLD
		);
	StChillerAlarms : 	STRUCT
		xNotRunning : BOOL; (*If we start chillerand dont recive the feedback*)
		xInAlarm : BOOL; (*ALarm directly from chiller*)
		xCheckChiller : BOOL; (*Alarm inform user to check chiller SP*)
		xAlrTempSensBrokn : BOOL; (*Chiller Heater Exchanger Sensor PT100 Borken or DIsconnected*)
		xAlrEnvTempSensBrokn : BOOL; (*Chiller Enviorenment Sensor PT100 Borken or DIsconnected*)
	END_STRUCT;
	StChillerOrders : 	STRUCT
		xRun : BOOL; (*Order to Start the Chiller*)
	END_STRUCT;
	StChillerComands : 	STRUCT
		xReset : BOOL; (*Reset Signal*)
		xMute : BOOL; (*Mute alarms sound*)
	END_STRUCT;
	StChillerStatusWaterManifold : 	STRUCT
		rEnviromentTemp : REAL;
		rManifoldTemp : REAL;
	END_STRUCT;
	StChillerStates : 	STRUCT
		xInstalled : BOOL; (*The system is or can be installed*)
		xEnabled : BOOL; (*The Chiller is enabled and raises alarms*)
		Status : ChillerStatus_enum;
		WaterManifold : StChillerStatusWaterManifold;
		xRunning : BOOL;
	END_STRUCT;
	StChillerSignalsOut : 	STRUCT
		xStart : BOOL; (*Start Chiller Out*)
	END_STRUCT;
	StChillerSignalsInWaterManifold : 	STRUCT
		iEnvironmentTempRaw : INT;
		iWaterManifoldTempRaw : INT;
		xTempEnvSensError : BOOL; (*Temperature enviorement sensor error*)
		xTempWatSensError : BOOL; (*Temperature water collector sensor error*)
	END_STRUCT;
	StChillerSignalsIn : 	STRUCT
		xCooling : BOOL; (*Chiller is cooling/running*)
		xPowered : BOOL; (*Chiller is powered on*)
		xAlarm : BOOL; (*Chiller is in alarm*)
		rSystemTemp : REAL; (*Temeperature of the system controlled by Chiller*)
		WaterManifold : StChillerSignalsInWaterManifold;
	END_STRUCT;
	StChillerParSw : 	STRUCT
		xEnable : BOOL; (*Enable the NonCrash in the machines where it can be installed*)
	END_STRUCT;
	StChillerParametersWaterManifold : 	STRUCT
		xSystemRunning : BOOL; (*The system to cool with the Chiller is started*)
	END_STRUCT;
	StChillerParameters : 	STRUCT
		xEnable : BOOL;
		xInstalled : BOOL; (*The system is or can be installed*)
		SystemType : ChillerSystemType_enum := CHILLERSYS_UNDEFINED;
		WaterManifold : StChillerParametersWaterManifold;
		rTempSetPoint : REAL; (*SetPoint Temperature*)
	END_STRUCT;
	StChiller : 	STRUCT
		AlSummary : stEFI_AlarmSummary;
		Alarm : StChillerAlarms;
		Orders : StChillerOrders;
		commands : StChillerComands;
		In : StChillerSignalsIn;
		Out : StChillerSignalsOut;
		St : StChillerStates;
		parSw : StChillerParSw;
		Parameters : StChillerParameters;
	END_STRUCT;
END_TYPE
```

### Program Logical/ExtPack/_Extras/ChillerCtrl/ChillerCtrl_v2/ChillerCtrl (IEC)

#### Conversions.st - Chiller control
```iecst
ACTION Conversions:

	CASE dataChill.Parameters.SystemType OF

		CHILLERSYS_DIRECT:

		CHILLERSYS_WATERMANIFOLD:
			dataChill.St.WaterManifold.rEnviromentTemp := INT_TO_REAL(dataChill.In.WaterManifold.iEnvironmentTempRaw)/10.0;
			dataChill.St.WaterManifold.rManifoldTemp := INT_TO_REAL(dataChill.In.WaterManifold.iWaterManifoldTempRaw)/10.0;

	END_CASE

END_ACTION
```

#### alarms.st - Chiller alarms
```iecst
ACTION alarms:

	//Reset Alarms with an external order to reset
	IF dataChill.commands.xReset THEN
		ResetAlarms;
	END_IF

	//Alarm: Chiller not running
	TON_DelayChillerNotRun.IN := dataChill.St.xRunning AND NOT dataChill.In.xPowered;
	TON_DelayChillerNotRun.PT := t#20s;
	TON_DelayChillerNotRun();

	IF TON_DelayChillerNotRun.Q THEN
		dataChill.Alarm.xNotRunning := TRUE;	//High Temperature Alarm Or not feedback
	END_IF

	//Alarm: Chiller in alarm
	TON_DelayChillerInAlarm.IN := dataChill.In.xAlarm;
	TON_DelayChillerInAlarm.PT := t#10s;
	TON_DelayChillerInAlarm();

	IF TON_DelayChillerInAlarm.Q THEN
		dataChill.Alarm.xInAlarm := TRUE;
	END_IF

	CASE dataChill.Parameters.SystemType OF

		CHILLERSYS_DIRECT:

		CHILLERSYS_WATERMANIFOLD:
			AlarmsWaterManifold;

	END_CASE

END_ACTION

ACTION ResetAlarms:
	dataChill.AlSummary:= stChillerAlarmsSummaryReseted;
	dataChill.Alarm:= stChillerAlarmsReseted;
END_ACTION

ACTION AlarmsWaterManifold:

	//Alarm: Chiller enviorenment temperature sensor error
	TON_DelayChillerEnvSensError.IN := dataChill.In.WaterManifold.xTempEnvSensError;
	TON_DelayChillerEnvSensError.PT := t#5s;
	TON_DelayChillerEnvSensError();

	IF TON_DelayChillerEnvSensError.Q THEN
		dataChill.Alarm.xAlrEnvTempSensBrokn := TRUE;
	END_IF

	//Alarm: Chiller water temperature sensor error
	TON_DelayChillerWatSensError.IN := dataChill.In.WaterManifold.xTempWatSensError;
	TON_DelayChillerWatSensError.PT := t#5s;
	TON_DelayChillerWatSensError();

	IF TON_DelayChillerWatSensError.Q THEN
		dataChill.Alarm.xAlrTempSensBrokn	:= TRUE;
	END_IF

	// show SP update message
	TON_DelayCheckChiller.IN := dataChill.St.xRunning;
	TON_DelayCheckChiller.PT := T#15m; //Time for the Chiller to arrive to Temperature
	TON_DelayCheckChiller();

	tonEstabCheck.IN := TON_DelayCheckChiller.Q AND (dataChill.Parameters.rTempSetPoint < dataChill.St.WaterManifold.rManifoldTemp);
	tonEstabCheck.PT := t#5s;
	tonEstabCheck();

	IF tonEstabCheck.Q THEN
		dataChill.Alarm.xCheckChiller := TRUE;
	END_IF

END_ACTION
```

#### alarmsSound.st - Chiller alarms sound
```iecst
ACTION alarmsSound:

	// Alarms reseteable sound management.
	ars_AlrStop.xAlarm:= dataChill.AlSummary.xAlarmStop;
	ars_AlrStop.xSilence:= dataChill.commands.xMute;
	ars_AlrStop();

	ars_AlrCritical.xAlarm:= dataChill.AlSummary.xAlarmCritical;
	ars_AlrCritical.xSilence:= dataChill.commands.xMute;
	ars_AlrCritical();

	ars_AlrWarning.xAlarm:= dataChill.AlSummary.xAnyWarning;
	ars_AlrWarning.xSilence:= dataChill.commands.xMute;
	ars_AlrWarning();

	dataChill.AlSummary.xAlarmSound:= 	//ars_AlrWarning.xAlarmSound OR
										ars_AlrStop.xAlarmSound OR
										ars_AlrCritical.xAlarmSound;

END_ACTION
```

#### alarmsSummary.st - Chiller alarms summary
```iecst
ACTION alarmsSummary:

	//Alarms Summary
	//Warning
	iReasonWarning.0 := dataChill.Alarm.xInAlarm;
	iReasonWarning.1 := dataChill.Alarm.xAlrEnvTempSensBrokn;
	iReasonWarning.2 := dataChill.Alarm.xAlrTempSensBrokn;
	iReasonWarning.3 := dataChill.Alarm.xNotRunning;
	iReasonWarning.4 := dataChill.Alarm.xCheckChiller;

	dataChill.AlSummary.xAnyWarning := iReasonWarning > 0;

	//Stop
	//iReasonStop.0 := ;
	dataChill.AlSummary.xAlarmStop := iReasonStop > 0;
	IF EDGEPOS(dataChill.AlSummary.xAlarmStop) THEN
		dataChill.AlSummary.iReasonStop[0] := iReasonStop;
		//LogStopAlarm;
	END_IF

	//Critical
	//iReasonCritical.0 := ;
	dataChill.AlSummary.xAlarmCritical:= iReasonCritical > 0;
	IF EDGEPOS(dataChill.AlSummary.xAlarmCritical) THEN
		dataChill.AlSummary.iReasonCritical := iReasonCritical;
		//LogCriticalAlarm;
	END_IF

END_ACTION
```

#### ChillerCtrl.var - Local variables
```iecst
VAR
	stChillerAlarmsReseted : StChillerAlarms;
	stChillerAlarmsSummaryReseted : stEFI_AlarmSummary;
	tonChillerOFF : TON;
	tonChillerON : TON;
	xNeedCold : BOOL;
	dataChill : REFERENCE TO StChiller;
	xEnoughCold : BOOL;
	TON_DelayChillerStopped : TON;
	TON_DelayChillerNotRun : TON;
END_VAR
VAR CONSTANT
	LC_OFFSET_TEMP_TO_START_STOP : REAL := 2.0; (*Temperature Offset to Start Chiller*)
END_VAR
VAR
	TON_DelayCheckChiller : TON; (*Time to delay check chiller message*)
	TON_DelayChillerEnvSensError : TON;
	TON_DelayChillerWatSensError : TON;
	TON_DelayChillerInAlarm : TON;
	tonEstabCheck : TON;
	ChillerState : ChillerStatus_enum;
	tonChillerRunning : TON;
	iReasonRunning : UINT;
	xManifoldRunOrder : BOOL;
	xRunOrder : BOOL;
	iReasonAlarm : USINT;
	iReasonSound : USINT;
	iReasonCritical : UDINT;
	iReasonWarning : UDINT;
	iReasonStop : UDINT;
	stEventLog : EventLog_typ;
	stEventLogCritical : EventLog_typ;
	ars_AlrWarning : AutoResetSound;
	ars_AlrStop : AutoResetSound;
	ars_AlrCritical : AutoResetSound;
END_VAR
```

- Program Logical/ExtPack/_Extras/ChillerCtrl/ChillerCtrl_v2/InitChiller (IEC) (no source held here)

### ChillerSim.typ - Local data types
```iecst
TYPE
	stChillerSimCommands : 	STRUCT
		StopRunning : BOOL;
		GenerateAlarm : BOOL;
	END_STRUCT;
	stChillerSim : 	STRUCT
		Commands : stChillerSimCommands;
	END_STRUCT;
END_TYPE
```

### ChillerSimGen.var - Local variables
```iecst
VAR
	iChillerSimIndex : USINT;
END_VAR
```

- Program Logical/ExtPack/_Extras/PowerMeterCtrl/PowerMeterCtrl_v1/InitPowerMeterCtrl (IEC) (no source held here)

### Program Logical/ExtPack/_Extras/PowerMeterCtrl/PowerMeterCtrl_v1/PowerMeterCtrl (IEC)

#### Alarms.st
```iecst
ACTION Alarms:

	//Saving modbus slave status when comms error raises
	IF EDGEPOS (PowerMeter.Alarms.xCommsError) THEN
		ModSlaveState := PowerMeter.Status.Comms.ModSlaveState;
		LastError := PowerMeter.Status.Comms.LastError;
		LastErrorBlockNum := PowerMeter.Status.Comms.LastErrorBlockNum;
	END_IF

	//Reset Alarms with an external order to reset
	IF PowerMeter.Commands.xReset THEN
		ResetAlarms;
	END_IF

	//Alarms related to comms
	IF NOT PowerMeter.Status.Comms.xModuleOk THEN
		PowerMeter.Alarms.xCommsError := TRUE;
	END_IF

END_ACTION

ACTION ResetAlarms:
	PowerMeter.Alarms := ResetedAlarms;
END_ACTION
```
